LIN {X 0,Y 162.203,Z 311.057,A -85,B 0,C 180,E1 -23302.53,E2 -23302.53} C_VEL
LIN {X 0,Y 161.888,Z 311.469,A -85,B 0,C 180,E1 -23307.51,E2 -23307.51} C_VEL
LIN {X 0,Y 161.935,Z 311.109,A -85,B 0,C 180,E1 -23309.998,E2 -23309.998} C_VEL
LIN {X 0,Y 162.113,Z 310.364,A -85,B 0,C 180,E1 -23312.483,E2 -23312.483} C_VEL
LIN {X 0,Y 162.905,Z 307.824,A -85,B 0,C 180,E1 -23317.126,E2 -23317.126} C_VEL
LIN {X 0,Y 164.1,Z 304.438,A -85,B 0,C 180,E1 -23321.109,E2 -23321.109} C_VEL
LIN {X 0,Y 165.769,Z 300.216,A -85,B 0,C 180,E1 -23324.734,E2 -23324.734} C_VEL
LIN {X 0,Y 168.468,Z 293.815,A -85,B 0,C 180,E1 -23328.86,E2 -23328.86} C_VEL
LIN {X 0,Y 171.418,Z 286.794,A -85,B 0,C 180,E1 -23332.283,E2 -23332.283} C_VEL
LIN {X 0,Y 174.792,Z 278.034,A -85,B 0,C 180,E1 -23335.606,E2 -23335.606} C_VEL
LIN {X 0,Y 178.001,Z 269.053,A -85,B 0,C 180,E1 -23338.277,E2 -23338.277} C_VEL
LIN {X 0,Y 179.645,Z 263.969,A -85,B 0,C 180,E1 -23339.551,E2 -23339.551} C_VEL
LIN {X 0,Y 179.703,Z 256.737,A -85,B 0,C 180,E1 -23341.534,E2 -23341.534} C_VEL
LIN {X 0,Y 178.862,Z 247.409,A -85,B 0,C 180,E1 -23343.952,E2 -23343.952} C_VEL
LIN {X 0,Y 177.345,Z 238.085,A -85,B 0,C 180,E1 -23346.202,E2 -23346.202} C_VEL
LIN {X 0,Y 174.11,Z 227.135,A -85,B 0,C 180,E1 -23348.872,E2 -23348.872} C_VEL
LIN {X 0,Y 169.319,Z 216.684,A -85,B 0,C 180,E1 -23351.656,E2 -23351.656} C_VEL
LIN {X 0,Y 167.341,Z 213.109,A -85,B 0,C 180,E1 -23352.687,E2 -23352.687} C_VEL
LIN {X 0,Y 166.28,Z 211.565,A -85,B 0,C 180,E1 -23353.185,E2 -23353.185} C_VEL
LIN {X 0,Y 164.764,Z 208.871,A -85,B 0,C 180,E1 -23353.961,E2 -23353.961} C_VEL
LIN {X 0,Y 164.403,Z 207.492,A -85,B 0,C 180,E1 -23354.271,E2 -23354.271} C_VEL
LIN {X 0,Y 164.349,Z 207.015,A -85,B 0,C 180,E1 -23356.826,E2 -23356.826} C_VEL
LIN {X 0,Y 164.334,Z 207.015,A -85,B 0,C 180,E1 -23360.328,E2 -23360.328} C_VEL
LIN {X 0,Y 164.319,Z 207.017,A -85,B 0,C 180,E1 -23366.218,E2 -23366.218} C_VEL
LIN {X 0,Y 164.376,Z 207.011,A -85,B 0,C 180,E1 -23369.131,E2 -23369.131} C_VEL
LIN {X 0,Y 164.404,Z 206.998,A -85,B 0,C 180,E1 -23374.691,E2 -23374.691} C_VEL
LIN {X 0,Y 164.507,Z 206.937,A -85,B 0,C 180,E1 -23380.014,E2 -23380.014} C_VEL
LIN {X 0,Y 164.546,Z 206.988,A -85,B 0,C 180,E1 -23385.151,E2 -23385.151} C_VEL
LIN {X 0,Y 164.838,Z 206.938,A -85,B 0,C 180,E1 -23390.18,E2 -23390.18} C_VEL
LIN {X 0,Y 164.846,Z 206.951,A -85,B 0,C 180,E1 -23392.651,E2 -23392.651} C_VEL
LIN {X 0,Y 165.029,Z 206.916,A -85,B 0,C 180,E1 -23397.559,E2 -23397.559} C_VEL
LIN {X 0,Y 165.272,Z 206.899,A -85,B 0,C 180,E1 -23399.999,E2 -23399.999} C_VEL
LIN {X 0,Y 164.763,Z 206.961,A -85,B 0,C 180,E1 -23404.893,E2 -23404.893} C_VEL
LIN {X 0,Y 164.833,Z 206.953,A -85,B 0,C 180,E1 -23407.348,E2 -23407.348} C_VEL
LIN {X 0,Y 164.725,Z 206.968,A -85,B 0,C 180,E1 -23411.13,E2 -23411.13} C_VEL
LIN {X 0,Y 164.485,Z 206.999,A -85,B 0,C 180,E1 -23417.403,E2 -23417.403} C_VEL
LIN {X 0,Y 164.506,Z 206.995,A -85,B 0,C 180,E1 -23419.985,E2 -23419.985} C_VEL
LIN {X 0,Y 164.379,Z 207.01,A -85,B 0,C 180,E1 -23426.135,E2 -23426.135} C_VEL
LIN {X 0,Y 164.37,Z 207.132,A -85,B 0,C 180,E1 -23431.687,E2 -23431.687} C_VEL
LIN {X 0,Y 164.77,Z 209.517,A -85,B 0,C 180,E1 -23436.665,E2 -23436.665} C_VEL
LIN {X 0,Y 165.051,Z 211.251,A -85,B 0,C 180,E1 -23439.971,E2 -23439.971} C_VEL
LIN {X 0,Y 165.48,Z 213.632,A -85,B 0,C 180,E1 -23444.186,E2 -23444.186} C_VEL
LIN {X 0,Y 166.572,Z 216.701,A -85,B 0,C 180,E1 -23444.816,E2 -23444.816} C_VEL
LIN {X 0,Y 168.249,Z 219.242,A -85,B 0,C 180,E1 -23445.593,E2 -23445.593} C_VEL
LIN {X 0,Y 170.168,Z 223.121,A -85,B 0,C 180,E1 -23446.592,E2 -23446.592} C_VEL
LIN {X 0,Y 173.545,Z 231.047,A -85,B 0,C 180,E1 -23448.52,E2 -23448.52} C_VEL
LIN {X 0,Y 175.71,Z 238.733,A -85,B 0,C 180,E1 -23450.216,E2 -23450.216} C_VEL
LIN {X 0,Y 177.253,Z 249.396,A -85,B 0,C 180,E1 -23452.465,E2 -23452.465} C_VEL
LIN {X 0,Y 177.858,Z 259.284,A -85,B 0,C 180,E1 -23454.703,E2 -23454.703} C_VEL
LIN {X 0,Y 177.686,Z 268.748,A -85,B 0,C 180,E1 -23457.058,E2 -23457.058} C_VEL
LIN {X 0,Y 176.797,Z 277.668,A -85,B 0,C 180,E1 -23459.551,E2 -23459.551} C_VEL
LIN {X 0,Y 173.444,Z 286.731,A -85,B 0,C 180,E1 -23462.23,E2 -23462.23} C_VEL
LIN {X 0,Y 170.179,Z 295.589,A -85,B 0,C 180,E1 -23465.612,E2 -23465.612} C_VEL
LIN {X 0,Y 167.31,Z 302.673,A -85,B 0,C 180,E1 -23469.084,E2 -23469.084} C_VEL
LIN {X 0,Y 164.995,Z 308.331,A -85,B 0,C 180,E1 -23472.655,E2 -23472.655} C_VEL
LIN {X 0,Y 163.395,Z 312.791,A -85,B 0,C 180,E1 -23476.319,E2 -23476.319} C_VEL
LIN {X 0,Y 162.403,Z 316.172,A -85,B 0,C 180,E1 -23480.034,E2 -23480.034} C_VEL
LIN {X 0,Y 161.999,Z 317.853,A -85,B 0,C 180,E1 -23482.524,E2 -23482.524} C_VEL
LIN {X 0,Y 161.79,Z 319.131,A -85,B 0,C 180,E1 -23485.018,E2 -23485.018} C_VEL
LIN {X 0,Y 161.765,Z 320.074,A -85,B 0,C 180,E1 -23487.78,E2 -23487.78} C_VEL
LIN {X 0,Y 161.896,Z 320.453,A -85,B 0,C 180,E1 -23490.002,E2 -23490.002} C_VEL
LIN {X 0,Y 161.765,Z 320.488,A -85,B 0,C 180,E1 -23492.492,E2 -23492.492} C_VEL
LIN {X 0,Y 161.791,Z 320.137,A -85,B 0,C 180,E1 -23494.985,E2 -23494.985} C_VEL
LIN {X 0,Y 162.002,Z 319.402,A -85,B 0,C 180,E1 -23497.479,E2 -23497.479} C_VEL
LIN {X 0,Y 162.416,Z 318.234,A -85,B 0,C 180,E1 -23499.968,E2 -23499.968} C_VEL
LIN {X 0,Y 163.497,Z 315.722,A -85,B 0,C 180,E1 -23503.676,E2 -23503.676} C_VEL
LIN {X 0,Y 165.117,Z 312.206,A -85,B 0,C 180,E1 -23507.335,E2 -23507.335} C_VEL
LIN {X 0,Y 167.532,Z 307.605,A -85,B 0,C 180,E1 -23510.89,E2 -23510.89} C_VEL
LIN {X 0,Y 171.01,Z 300.727,A -85,B 0,C 180,E1 -23514.869,E2 -23514.869} C_VEL
LIN {X 0,Y 174.459,Z 293.132,A -85,B 0,C 180,E1 -23518.251,E2 -23518.251} C_VEL
LIN {X 0,Y 178.393,Z 284.443,A -85,B 0,C 180,E1 -23521.198,E2 -23521.198} C_VEL
LIN {X 0,Y 179.136,Z 281.733,A -85,B 0,C 180,E1 -23522.062,E2 -23522.062} C_VEL
LIN {X 0,Y 178.984,Z 277.803,A -85,B 0,C 180,E1 -23523.47,E2 -23523.47} C_VEL
LIN {X 0,Y 177.92,Z 274.075,A -85,B 0,C 180,E1 -23524.927,E2 -23524.927} C_VEL
LIN {X 0,Y 175.412,Z 266.243,A -85,B 0,C 180,E1 -23527.891,E2 -23527.891} C_VEL
LIN {X 0,Y 175.084,Z 263.3,A -85,B 0,C 180,E1 -23528.808,E2 -23528.808} C_VEL
LIN {X 0,Y 174.738,Z 253.125,A -85,B 0,C 180,E1 -23531.496,E2 -23531.496} C_VEL
LIN {X 0,Y 173.737,Z 246.452,A -85,B 0,C 180,E1 -23533.27,E2 -23533.27} C_VEL
LIN {X 0,Y 171.827,Z 240.22,A -85,B 0,C 180,E1 -23535.125,E2 -23535.125} C_VEL
LIN {X 0,Y 168.637,Z 232.567,A -85,B 0,C 180,E1 -23537.626,E2 -23537.626} C_VEL
LIN {X 0,Y 166.729,Z 228.56,A -85,B 0,C 180,E1 -23539.007,E2 -23539.007} C_VEL
LIN {X 0,Y 164.338,Z 223.902,A -85,B 0,C 180,E1 -23540.694,E2 -23540.694} C_VEL
LIN {X 0,Y 162.287,Z 220.406,A -85,B 0,C 180,E1 -23542.092,E2 -23542.092} C_VEL
LIN {X 0,Y 161.446,Z 218.634,A -85,B 0,C 180,E1 -23542.707,E2 -23542.707} C_VEL
LIN {X 0,Y 159.069,Z 215.483,A -85,B 0,C 180,E1 -23544.252,E2 -23544.252} C_VEL
LIN {X 0,Y 158.095,Z 212.845,A -85,B 0,C 180,E1 -23545.087,E2 -23545.087} C_VEL
LIN {X 0,Y 157.947,Z 211.689,A -85,B 0,C 180,E1 -23547.728,E2 -23547.728} C_VEL
LIN {X 0,Y 157.59,Z 209.431,A -85,B 0,C 180,E1 -23553.515,E2 -23553.515} C_VEL
LIN {X 0,Y 157.415,Z 208.47,A -85,B 0,C 180,E1 -23556.309,E2 -23556.309} C_VEL
LIN {X 0,Y 157.441,Z 207.873,A -85,B 0,C 180,E1 -23559.616,E2 -23559.616} C_VEL
LIN {X 0,Y 157.456,Z 207.873,A -85,B 0,C 180,E1 -23564.467,E2 -23564.467} C_VEL
LIN {X 0,Y 157.681,Z 207.842,A -85,B 0,C 180,E1 -23569.731,E2 -23569.731} C_VEL
LIN {X 0,Y 157.758,Z 207.832,A -85,B 0,C 180,E1 -23572.32,E2 -23572.32} C_VEL
LIN {X 0,Y 158.242,Z 207.772,A -85,B 0,C 180,E1 -23580.001,E2 -23580.001} C_VEL
LIN {X 0,Y 157.711,Z 207.84,A -85,B 0,C 180,E1 -23585.114,E2 -23585.114} C_VEL
LIN {X 0,Y 157.756,Z 207.835,A -85,B 0,C 180,E1 -23587.681,E2 -23587.681} C_VEL
LIN {X 0,Y 157.626,Z 207.85,A -85,B 0,C 180,E1 -23591.227,E2 -23591.227} C_VEL
LIN {X 0,Y 157.431,Z 207.873,A -85,B 0,C 180,E1 -23595.537,E2 -23595.537} C_VEL
LIN {X 0,Y 157.364,Z 207.884,A -85,B 0,C 180,E1 -23600.934,E2 -23600.934} C_VEL
LIN {X 0,Y 157.306,Z 207.889,A -85,B 0,C 180,E1 -23606.682,E2 -23606.682} C_VEL
LIN {X 0,Y 157.312,Z 208.05,A -85,B 0,C 180,E1 -23611.918,E2 -23611.918} C_VEL
LIN {X 0,Y 157.324,Z 208.308,A -85,B 0,C 180,E1 -23612.607,E2 -23612.607} C_VEL
LIN {X 0,Y 158.283,Z 210.846,A -85,B 0,C 180,E1 -23613.427,E2 -23613.427} C_VEL
LIN {X 0,Y 160.753,Z 213.678,A -85,B 0,C 180,E1 -23615.039,E2 -23615.039} C_VEL
LIN {X 0,Y 163.069,Z 217.809,A -85,B 0,C 180,E1 -23616.717,E2 -23616.717} C_VEL
LIN {X 0,Y 164.239,Z 219.482,A -85,B 0,C 180,E1 -23617.478,E2 -23617.478} C_VEL
LIN {X 0,Y 166.404,Z 223.337,A -85,B 0,C 180,E1 -23619.019,E2 -23619.019} C_VEL
LIN {X 0,Y 171.596,Z 234.254,A -85,B 0,C 180,E1 -23622.965,E2 -23622.965} C_VEL
LIN {X 0,Y 173.907,Z 240.964,A -85,B 0,C 180,E1 -23625.142,E2 -23625.142} C_VEL
LIN {X 0,Y 175.503,Z 248.167,A -85,B 0,C 180,E1 -23627.335,E2 -23627.335} C_VEL
LIN {X 0,Y 176.566,Z 257.323,A -85,B 0,C 180,E1 -23630.091,E2 -23630.091} C_VEL
LIN {X 0,Y 176.728,Z 265.588,A -85,B 0,C 180,E1 -23632.689,E2 -23632.689} C_VEL
LIN {X 0,Y 176.42,Z 269.664,A -85,B 0,C 180,E1 -23634.015,E2 -23634.015} C_VEL
LIN {X 0,Y 172.646,Z 278.623,A -85,B 0,C 180,E1 -23636.664,E2 -23636.664} C_VEL
LIN {X 0,Y 168.441,Z 287.36,A -85,B 0,C 180,E1 -23639.955,E2 -23639.955} C_VEL
LIN {X 0,Y 164.622,Z 294.525,A -85,B 0,C 180,E1 -23643.505,E2 -23643.505} C_VEL
LIN {X 0,Y 161.73,Z 299.883,A -85,B 0,C 180,E1 -23646.977,E2 -23646.977} C_VEL
LIN {X 0,Y 159.205,Z 304.249,A -85,B 0,C 180,E1 -23650.665,E2 -23650.665} C_VEL
LIN {X 0,Y 157.287,Z 307.544,A -85,B 0,C 180,E1 -23654.448,E2 -23654.448} C_VEL
LIN {X 0,Y 155.652,Z 310.41,A -85,B 0,C 180,E1 -23659.594,E2 -23659.594} C_VEL
LIN {X 0,Y 155.167,Z 311.244,A -85,B 0,C 180,E1 -23662.189,E2 -23662.189} C_VEL
LIN {X 0,Y 154.798,Z 311.67,A -85,B 0,C 180,E1 -23667.396,E2 -23667.396} C_VEL
LIN {X 0,Y 154.835,Z 311.316,A -85,B 0,C 180,E1 -23669.998,E2 -23669.998} C_VEL
LIN {X 0,Y 155.035,Z 310.579,A -85,B 0,C 180,E1 -23672.596,E2 -23672.596} C_VEL
LIN {X 0,Y 155.736,Z 308.452,A -85,B 0,C 180,E1 -23676.869,E2 -23676.869} C_VEL
LIN {X 0,Y 157.159,Z 304.68,A -85,B 0,C 180,E1 -23681.607,E2 -23681.607} C_VEL
LIN {X 0,Y 158.921,Z 300.471,A -85,B 0,C 180,E1 -23685.384,E2 -23685.384} C_VEL
LIN {X 0,Y 161.764,Z 294.086,A -85,B 0,C 180,E1 -23689.673,E2 -23689.673} C_VEL
LIN {X 0,Y 164.871,Z 287.089,A -85,B 0,C 180,E1 -23693.219,E2 -23693.219} C_VEL
LIN {X 0,Y 168.434,Z 278.348,A -85,B 0,C 180,E1 -23696.647,E2 -23696.647} C_VEL
LIN {X 0,Y 171.792,Z 269.391,A -85,B 0,C 180,E1 -23699.397,E2 -23699.397} C_VEL
LIN {X 0,Y 173.31,Z 264.918,A -85,B 0,C 180,E1 -23700.556,E2 -23700.556} C_VEL
LIN {X 0,Y 173.334,Z 256.195,A -85,B 0,C 180,E1 -23703.096,E2 -23703.096} C_VEL
LIN {X 0,Y 172.301,Z 245.415,A -85,B 0,C 180,E1 -23706.01,E2 -23706.01} C_VEL
LIN {X 0,Y 170.636,Z 237.194,A -85,B 0,C 180,E1 -23708.151,E2 -23708.151} C_VEL
LIN {X 0,Y 168.166,Z 229.23,A -85,B 0,C 180,E1 -23710.296,E2 -23710.296} C_VEL
LIN {X 0,Y 163.955,Z 220.22,A -85,B 0,C 180,E1 -23712.995,E2 -23712.995} C_VEL
LIN {X 0,Y 162.101,Z 216.724,A -85,B 0,C 180,E1 -23714.084,E2 -23714.084} C_VEL
LIN {X 0,Y 160.266,Z 213.131,A -85,B 0,C 180,E1 -23715.181,E2 -23715.181} C_VEL
LIN {X 0,Y 157.998,Z 210.26,A -85,B 0,C 180,E1 -23716.352,E2 -23716.352} C_VEL
LIN {X 0,Y 157.297,Z 207.894,A -85,B 0,C 180,E1 -23716.889,E2 -23716.889} C_VEL
LIN {X 0,Y 157.252,Z 207.899,A -85,B 0,C 180,E1 -23721.266,E2 -23721.266} C_VEL
LIN {X 0,Y 157.278,Z 207.892,A -85,B 0,C 180,E1 -23724.485,E2 -23724.485} C_VEL
LIN {X 0,Y 157.282,Z 207.89,A -85,B 0,C 180,E1 -23728.093,E2 -23728.093} C_VEL
LIN {X 0,Y 157.308,Z 207.89,A -85,B 0,C 180,E1 -23733.463,E2 -23733.463} C_VEL
LIN {X 0,Y 157.433,Z 207.815,A -85,B 0,C 180,E1 -23739.614,E2 -23739.614} C_VEL
LIN {X 0,Y 157.474,Z 207.865,A -85,B 0,C 180,E1 -23744.467,E2 -23744.467} C_VEL
LIN {X 0,Y 157.757,Z 207.818,A -85,B 0,C 180,E1 -23749.735,E2 -23749.735} C_VEL
LIN {X 0,Y 157.808,Z 207.828,A -85,B 0,C 180,E1 -23752.321,E2 -23752.321} C_VEL
LIN {X 0,Y 158.235,Z 207.775,A -85,B 0,C 180,E1 -23759.999,E2 -23759.999} C_VEL
LIN {X 0,Y 157.712,Z 207.84,A -85,B 0,C 180,E1 -23765.113,E2 -23765.113} C_VEL
LIN {X 0,Y 157.79,Z 207.832,A -85,B 0,C 180,E1 -23767.678,E2 -23767.678} C_VEL
LIN {X 0,Y 157.656,Z 207.848,A -85,B 0,C 180,E1 -23771.299,E2 -23771.299} C_VEL
LIN {X 0,Y 157.443,Z 207.876,A -85,B 0,C 180,E1 -23775.535,E2 -23775.535} C_VEL
LIN {X 0,Y 157.401,Z 207.879,A -85,B 0,C 180,E1 -23780.928,E2 -23780.928} C_VEL
LIN {X 0,Y 157.301,Z 207.89,A -85,B 0,C 180,E1 -23786.686,E2 -23786.686} C_VEL
LIN {X 0,Y 157.31,Z 207.905,A -85,B 0,C 180,E1 -23790.08,E2 -23790.08} C_VEL
LIN {X 0,Y 157.7,Z 210.271,A -85,B 0,C 180,E1 -23795.405,E2 -23795.405} C_VEL
LIN {X 0,Y 158.195,Z 213.385,A -85,B 0,C 180,E1 -23801.502,E2 -23801.502} C_VEL
LIN {X 0,Y 159.386,Z 216.528,A -85,B 0,C 180,E1 -23802.255,E2 -23802.255} C_VEL
LIN {X 0,Y 161.229,Z 219.165,A -85,B 0,C 180,E1 -23803.199,E2 -23803.199} C_VEL
LIN {X 0,Y 163.297,Z 223.265,A -85,B 0,C 180,E1 -23804.393,E2 -23804.393} C_VEL
LIN {X 0,Y 166.774,Z 230.949,A -85,B 0,C 180,E1 -23806.52,E2 -23806.52} C_VEL
LIN {X 0,Y 169.541,Z 239.112,A -85,B 0,C 180,E1 -23808.62,E2 -23808.62} C_VEL
LIN {X 0,Y 170.958,Z 248.36,A -85,B 0,C 180,E1 -23810.71,E2 -23810.71} C_VEL
LIN {X 0,Y 171.59,Z 258.978,A -85,B 0,C 180,E1 -23813.236,E2 -23813.236} C_VEL
LIN {X 0,Y 171.422,Z 268.343,A -85,B 0,C 180,E1 -23815.681,E2 -23815.681} C_VEL
LIN {X 0,Y 170.445,Z 277.327,A -85,B 0,C 180,E1 -23818.287,E2 -23818.287} C_VEL
LIN {X 0,Y 168.499,Z 283,A -85,B 0,C 180,E1 -23819.97,E2 -23819.97} C_VEL
LIN {X 0,Y 165.319,Z 291.103,A -85,B 0,C 180,E1 -23822.811,E2 -23822.811} C_VEL
LIN {X 0,Y 162.159,Z 299.059,A -85,B 0,C 180,E1 -23826.369,E2 -23826.369} C_VEL
LIN {X 0,Y 159.836,Z 304.439,A -85,B 0,C 180,E1 -23829.408,E2 -23829.408} C_VEL
LIN {X 0,Y 157.544,Z 309.705,A -85,B 0,C 180,E1 -23833.147,E2 -23833.147} C_VEL
LIN {X 0,Y 156.046,Z 313.804,A -85,B 0,C 180,E1 -23836.989,E2 -23836.989} C_VEL
LIN {X 0,Y 155.406,Z 315.944,A -85,B 0,C 180,E1 -23839.581,E2 -23839.581} C_VEL
LIN {X 0,Y 154.948,Z 317.631,A -85,B 0,C 180,E1 -23842.182,E2 -23842.182} C_VEL
LIN {X 0,Y 154.71,Z 318.914,A -85,B 0,C 180,E1 -23844.789,E2 -23844.789} C_VEL
LIN {X 0,Y 154.683,Z 319.986,A -85,B 0,C 180,E1 -23848.307,E2 -23848.307} C_VEL
LIN {X 0,Y 154.794,Z 320.253,A -85,B 0,C 180,E1 -23850.002,E2 -23850.002} C_VEL
LIN {X 0,Y 154.69,Z 320.293,A -85,B 0,C 180,E1 -23852.606,E2 -23852.606} C_VEL
LIN {X 0,Y 154.952,Z 319.218,A -85,B 0,C 180,E1 -23857.822,E2 -23857.822} C_VEL
LIN {X 0,Y 155.418,Z 318.06,A -85,B 0,C 180,E1 -23860.422,E2 -23860.422} C_VEL
LIN {X 0,Y 156.133,Z 316.478,A -85,B 0,C 180,E1 -23863.007,E2 -23863.007} C_VEL
LIN {X 0,Y 157.659,Z 313.312,A -85,B 0,C 180,E1 -23866.844,E2 -23866.844} C_VEL
LIN {X 0,Y 159.989,Z 309.096,A -85,B 0,C 180,E1 -23870.575,E2 -23870.575} C_VEL
LIN {X 0,Y 162.92,Z 303.71,A -85,B 0,C 180,E1 -23874.193,E2 -23874.193} C_VEL
LIN {X 0,Y 166.299,Z 296.973,A -85,B 0,C 180,E1 -23877.702,E2 -23877.702} C_VEL
LIN {X 0,Y 170.363,Z 288.626,A -85,B 0,C 180,E1 -23881.041,E2 -23881.041} C_VEL
LIN {X 0,Y 173.344,Z 281.875,A -85,B 0,C 180,E1 -23883.184,E2 -23883.184} C_VEL
LIN {X 0,Y 174.641,Z 273.581,A -85,B 0,C 180,E1 -23885.819,E2 -23885.819} C_VEL
LIN {X 0,Y 175.094,Z 264.082,A -85,B 0,C 180,E1 -23888.583,E2 -23888.583} C_VEL
LIN {X 0,Y 175.084,Z 263.3,A -85,B 0,C 180,E1 -23888.808,E2 -23888.808} C_VEL
LIN {X 0,Y 174.426,Z 259.081,A -85,B 0,C 180,E1 -23890.152,E2 -23890.152} C_VEL
LIN {X 0,Y 172.876,Z 255.276,A -85,B 0,C 180,E1 -23891.575,E2 -23891.575} C_VEL
LIN {X 0,Y 168.701,Z 248.158,A -85,B 0,C 180,E1 -23894.542,E2 -23894.542} C_VEL
LIN {X 0,Y 166.316,Z 242.998,A -85,B 0,C 180,E1 -23896.51,E2 -23896.51} C_VEL
LIN {X 0,Y 162.824,Z 234.197,A -85,B 0,C 180,E1 -23899.651,E2 -23899.651} C_VEL
LIN {X 0,Y 159.954,Z 228.545,A -85,B 0,C 180,E1 -23901.939,E2 -23901.939} C_VEL
LIN {X 0,Y 157.693,Z 224.076,A -85,B 0,C 180,E1 -23903.785,E2 -23903.785} C_VEL
LIN {X 0,Y 155.296,Z 220.209,A -85,B 0,C 180,E1 -23905.648,E2 -23905.648} C_VEL
LIN {X 0,Y 154.514,Z 218.494,A -85,B 0,C 180,E1 -23906.335,E2 -23906.335} C_VEL
LIN {X 0,Y 152.056,Z 215.517,A -85,B 0,C 180,E1 -23908.204,E2 -23908.204} C_VEL
LIN {X 0,Y 150.93,Z 212.808,A -85,B 0,C 180,E1 -23909.286,E2 -23909.286} C_VEL
LIN {X 0,Y 150.85,Z 212.305,A -85,B 0,C 180,E1 -23909.945,E2 -23909.945} C_VEL
LIN {X 0,Y 150.531,Z 210.458,A -85,B 0,C 180,E1 -23915.154,E2 -23915.154} C_VEL
LIN {X 0,Y 150.387,Z 208.751,A -85,B 0,C 180,E1 -23920.906,E2 -23920.906} C_VEL
LIN {X 0,Y 150.432,Z 208.748,A -85,B 0,C 180,E1 -23926.492,E2 -23926.492} C_VEL
LIN {X 0,Y 150.604,Z 208.726,A -85,B 0,C 180,E1 -23929.243,E2 -23929.243} C_VEL
LIN {X 0,Y 150.695,Z 208.713,A -85,B 0,C 180,E1 -23931.958,E2 -23931.958} C_VEL
LIN {X 0,Y 151.204,Z 208.649,A -85,B 0,C 180,E1 -23940.001,E2 -23940.001} C_VEL
LIN {X 0,Y 150.64,Z 208.716,A -85,B 0,C 180,E1 -23946.982,E2 -23946.982} C_VEL
LIN {X 0,Y 150.568,Z 208.728,A -85,B 0,C 180,E1 -23951.43,E2 -23951.43} C_VEL
LIN {X 0,Y 150.343,Z 208.758,A -85,B 0,C 180,E1 -23956.289,E2 -23956.289} C_VEL
LIN {X 0,Y 150.346,Z 208.758,A -85,B 0,C 180,E1 -23960.792,E2 -23960.792} C_VEL
LIN {X 0,Y 150.238,Z 208.771,A -85,B 0,C 180,E1 -23967.281,E2 -23967.281} C_VEL
LIN {X 0,Y 150.203,Z 208.777,A -85,B 0,C 180,E1 -23968.279,E2 -23968.279} C_VEL
LIN {X 0,Y 150.914,Z 211.097,A -85,B 0,C 180,E1 -23969.084,E2 -23969.084} C_VEL
LIN {X 0,Y 152.923,Z 213.602,A -85,B 0,C 180,E1 -23970.723,E2 -23970.723} C_VEL
LIN {X 0,Y 154.214,Z 214.632,A -85,B 0,C 180,E1 -23971.641,E2 -23971.641} C_VEL
LIN {X 0,Y 156.009,Z 218.019,A -85,B 0,C 180,E1 -23973.205,E2 -23973.205} C_VEL
LIN {X 0,Y 157.587,Z 220.032,A -85,B 0,C 180,E1 -23974.364,E2 -23974.364} C_VEL
LIN {X 0,Y 159.667,Z 223.754,A -85,B 0,C 180,E1 -23976.067,E2 -23976.067} C_VEL
LIN {X 0,Y 163.659,Z 231.631,A -85,B 0,C 180,E1 -23979.381,E2 -23979.381} C_VEL
LIN {X 0,Y 166.926,Z 239.317,A -85,B 0,C 180,E1 -23982.35,E2 -23982.35} C_VEL
LIN {X 0,Y 169.117,Z 247.172,A -85,B 0,C 180,E1 -23985.054,E2 -23985.054} C_VEL
LIN {X 0,Y 170.207,Z 254.802,A -85,B 0,C 180,E1 -23987.505,E2 -23987.505} C_VEL
LIN {X 0,Y 170.646,Z 263.364,A -85,B 0,C 180,E1 -23990.333,E2 -23990.333} C_VEL
LIN {X 0,Y 170.321,Z 270.371,A -85,B 0,C 180,E1 -23992.758,E2 -23992.758} C_VEL
LIN {X 0,Y 167.564,Z 277.078,A -85,B 0,C 180,E1 -23994.782,E2 -23994.782} C_VEL
LIN {X 0,Y 163.02,Z 286.111,A -85,B 0,C 180,E1 -23998.123,E2 -23998.123} C_VEL
LIN {X 0,Y 158.942,Z 293.494,A -85,B 0,C 180,E1 -24001.691,E2 -24001.691} C_VEL
LIN {X 0,Y 155.173,Z 300.024,A -85,B 0,C 180,E1 -24005.944,E2 -24005.944} C_VEL
LIN {X 0,Y 152.509,Z 304.402,A -85,B 0,C 180,E1 -24009.78,E2 -24009.78} C_VEL
LIN {X 0,Y 150.432,Z 307.711,A -85,B 0,C 180,E1 -24013.72,E2 -24013.72} C_VEL
LIN {X 0,Y 148.664,Z 310.588,A -85,B 0,C 180,E1 -24019.099,E2 -24019.099} C_VEL
LIN {X 0,Y 148.113,Z 311.431,A -85,B 0,C 180,E1 -24021.815,E2 -24021.815} C_VEL
LIN {X 0,Y 147.718,Z 311.87,A -85,B 0,C 180,E1 -24027.271,E2 -24027.271} C_VEL
LIN {X 0,Y 147.748,Z 311.522,A -85,B 0,C 180,E1 -24029.998,E2 -24029.998} C_VEL
LIN {X 0,Y 147.946,Z 310.793,A -85,B 0,C 180,E1 -24032.721,E2 -24032.721} C_VEL
LIN {X 0,Y 148.54,Z 309.074,A -85,B 0,C 180,E1 -24036.482,E2 -24036.482} C_VEL
LIN {X 0,Y 150.216,Z 304.922,A -85,B 0,C 180,E1 -24042.151,E2 -24042.151} C_VEL
LIN {X 0,Y 152.105,Z 300.727,A -85,B 0,C 180,E1 -24046.092,E2 -24046.092} C_VEL
LIN {X 0,Y 155.096,Z 294.356,A -85,B 0,C 180,E1 -24050.556,E2 -24050.556} C_VEL
LIN {X 0,Y 158.382,Z 287.384,A -85,B 0,C 180,E1 -24054.23,E2 -24054.23} C_VEL
LIN {X 0,Y 162.115,Z 278.664,A -85,B 0,C 180,E1 -24057.773,E2 -24057.773} C_VEL
LIN {X 0,Y 165.656,Z 269.729,A -85,B 0,C 180,E1 -24060.6,E2 -24060.6} C_VEL
LIN {X 0,Y 166.986,Z 265.869,A -85,B 0,C 180,E1 -24061.647,E2 -24061.647} C_VEL
LIN {X 0,Y 167.052,Z 255.964,A -85,B 0,C 180,E1 -24064.697,E2 -24064.697} C_VEL
LIN {X 0,Y 166.044,Z 245.62,A -85,B 0,C 180,E1 -24067.66,E2 -24067.66} C_VEL
LIN {X 0,Y 163.914,Z 236.216,A -85,B 0,C 180,E1 -24070.346,E2 -24070.346} C_VEL
LIN {X 0,Y 160.826,Z 228.089,A -85,B 0,C 180,E1 -24072.875,E2 -24072.875} C_VEL
LIN {X 0,Y 157.75,Z 221.69,A -85,B 0,C 180,E1 -24075.027,E2 -24075.027} C_VEL
LIN {X 0,Y 155.572,Z 217.717,A -85,B 0,C 180,E1 -24076.454,E2 -24076.454} C_VEL
LIN {X 0,Y 153.648,Z 214.551,A -85,B 0,C 180,E1 -24077.682,E2 -24077.682} C_VEL
LIN {X 0,Y 153.02,Z 213.601,A -85,B 0,C 180,E1 -24078.069,E2 -24078.069} C_VEL
LIN {X 0,Y 150.999,Z 211.254,A -85,B 0,C 180,E1 -24079.24,E2 -24079.24} C_VEL
LIN {X 0,Y 150.194,Z 208.776,A -85,B 0,C 180,E1 -24079.953,E2 -24079.953} C_VEL
LIN {X 0,Y 150.21,Z 208.773,A -85,B 0,C 180,E1 -24082.684,E2 -24082.684} C_VEL
LIN {X 0,Y 150.205,Z 208.771,A -85,B 0,C 180,E1 -24087.364,E2 -24087.364} C_VEL
LIN {X 0,Y 150.232,Z 208.772,A -85,B 0,C 180,E1 -24092.716,E2 -24092.716} C_VEL
LIN {X 0,Y 150.377,Z 208.691,A -85,B 0,C 180,E1 -24099.167,E2 -24099.167} C_VEL
LIN {X 0,Y 150.383,Z 208.74,A -85,B 0,C 180,E1 -24103.715,E2 -24103.715} C_VEL
LIN {X 0,Y 150.674,Z 208.699,A -85,B 0,C 180,E1 -24109.246,E2 -24109.246} C_VEL
LIN {X 0,Y 150.747,Z 208.705,A -85,B 0,C 180,E1 -24111.959,E2 -24111.959} C_VEL
LIN {X 0,Y 151.196,Z 208.652,A -85,B 0,C 180,E1 -24119.999,E2 -24119.999} C_VEL
LIN {X 0,Y 150.661,Z 208.719,A -85,B 0,C 180,E1 -24125.353,E2 -24125.353} C_VEL
LIN {X 0,Y 150.725,Z 208.712,A -85,B 0,C 180,E1 -24128.041,E2 -24128.041} C_VEL
LIN {X 0,Y 150.59,Z 208.728,A -85,B 0,C 180,E1 -24131.488,E2 -24131.488} C_VEL
LIN {X 0,Y 150.356,Z 208.757,A -85,B 0,C 180,E1 -24136.287,E2 -24136.287} C_VEL
LIN {X 0,Y 150.376,Z 208.754,A -85,B 0,C 180,E1 -24140.832,E2 -24140.832} C_VEL
LIN {X 0,Y 150.231,Z 208.772,A -85,B 0,C 180,E1 -24147.283,E2 -24147.283} C_VEL
LIN {X 0,Y 150.206,Z 208.847,A -85,B 0,C 180,E1 -24148.658,E2 -24148.658} C_VEL
LIN {X 0,Y 150.547,Z 210.529,A -85,B 0,C 180,E1 -24152.839,E2 -24152.839} C_VEL
LIN {X 0,Y 150.92,Z 213.026,A -85,B 0,C 180,E1 -24158.364,E2 -24158.364} C_VEL
LIN {X 0,Y 152.106,Z 216.252,A -85,B 0,C 180,E1 -24159.253,E2 -24159.253} C_VEL
LIN {X 0,Y 154.222,Z 219.149,A -85,B 0,C 180,E1 -24160.477,E2 -24160.477} C_VEL
LIN {X 0,Y 156.099,Z 222.817,A -85,B 0,C 180,E1 -24161.699,E2 -24161.699} C_VEL
LIN {X 0,Y 157.354,Z 225.261,A -85,B 0,C 180,E1 -24162.496,E2 -24162.496} C_VEL
LIN {X 0,Y 160.945,Z 232.932,A -85,B 0,C 180,E1 -24164.941,E2 -24164.941} C_VEL
LIN {X 0,Y 163.837,Z 241.739,A -85,B 0,C 180,E1 -24167.412,E2 -24167.412} C_VEL
LIN {X 0,Y 165.07,Z 250.965,A -85,B 0,C 180,E1 -24169.7,E2 -24169.7} C_VEL
LIN {X 0,Y 165.418,Z 261.952,A -85,B 0,C 180,E1 -24172.518,E2 -24172.518} C_VEL
LIN {X 0,Y 164.895,Z 271.574,A -85,B 0,C 180,E1 -24175.246,E2 -24175.246} C_VEL
LIN {X 0,Y 163.785,Z 278.967,A -85,B 0,C 180,E1 -24177.567,E2 -24177.567} C_VEL
LIN {X 0,Y 160.288,Z 287.755,A -85,B 0,C 180,E1 -24180.449,E2 -24180.449} C_VEL
LIN {X 0,Y 156.893,Z 295.84,A -85,B 0,C 180,E1 -24183.84,E2 -24183.84} C_VEL
LIN {X 0,Y 154.025,Z 302.14,A -85,B 0,C 180,E1 -24187.183,E2 -24187.183} C_VEL
LIN {X 0,Y 151.473,Z 307.829,A -85,B 0,C 180,E1 -24191.051,E2 -24191.051} C_VEL
LIN {X 0,Y 149.57,Z 312.312,A -85,B 0,C 180,E1 -24195.026,E2 -24195.026} C_VEL
LIN {X 0,Y 148.39,Z 315.716,A -85,B 0,C 180,E1 -24199.082,E2 -24199.082} C_VEL
LIN {X 0,Y 147.898,Z 317.409,A -85,B 0,C 180,E1 -24201.807,E2 -24201.807} C_VEL
LIN {X 0,Y 147.633,Z 318.698,A -85,B 0,C 180,E1 -24204.539,E2 -24204.539} C_VEL
LIN {X 0,Y 147.612,Z 319.908,A -85,B 0,C 180,E1 -24208.946,E2 -24208.946} C_VEL
LIN {X 0,Y 147.606,Z 320.098,A -85,B 0,C 180,E1 -24212.731,E2 -24212.731} C_VEL
LIN {X 0,Y 147.902,Z 319.033,A -85,B 0,C 180,E1 -24218.197,E2 -24218.197} C_VEL
LIN {X 0,Y 148.406,Z 317.885,A -85,B 0,C 180,E1 -24220.92,E2 -24220.92} C_VEL
LIN {X 0,Y 149.179,Z 316.309,A -85,B 0,C 180,E1 -24223.625,E2 -24223.625} C_VEL
LIN {X 0,Y 150.86,Z 313.155,A -85,B 0,C 180,E1 -24227.627,E2 -24227.627} C_VEL
LIN {X 0,Y 153.348,Z 308.951,A -85,B 0,C 180,E1 -24231.509,E2 -24231.509} C_VEL
LIN {X 0,Y 156.472,Z 303.578,A -85,B 0,C 180,E1 -24235.258,E2 -24235.258} C_VEL
LIN {X 0,Y 160.028,Z 296.855,A -85,B 0,C 180,E1 -24238.887,E2 -24238.887} C_VEL
LIN {X 0,Y 164.301,Z 288.529,A -85,B 0,C 180,E1 -24242.322,E2 -24242.322} C_VEL
LIN {X 0,Y 166.689,Z 283.578,A -85,B 0,C 180,E1 -24243.962,E2 -24243.962} C_VEL
LIN {X 0,Y 167.946,Z 278.002,A -85,B 0,C 180,E1 -24245.862,E2 -24245.862} C_VEL
LIN {X 0,Y 168.887,Z 269.391,A -85,B 0,C 180,E1 -24248.623,E2 -24248.623} C_VEL
LIN {X 0,Y 169.119,Z 258.96,A -85,B 0,C 180,E1 -24251.674,E2 -24251.674} C_VEL
LIN {X 0,Y 168.49,Z 251.064,A -85,B 0,C 180,E1 -24253.912,E2 -24253.912} C_VEL
LIN {X 0,Y 166.844,Z 244.583,A -85,B 0,C 180,E1 -24255.969,E2 -24255.969} C_VEL
LIN {X 0,Y 166.316,Z 242.998,A -85,B 0,C 180,E1 -24256.51,E2 -24256.51} C_VEL
LIN {X 0,Y 164.51,Z 239.362,A -85,B 0,C 180,E1 -24257.99,E2 -24257.99} C_VEL
LIN {X 0,Y 162.082,Z 236.448,A -85,B 0,C 180,E1 -24259.589,E2 -24259.589} C_VEL
LIN {X 0,Y 153.126,Z 228.349,A -85,B 0,C 180,E1 -24265.436,E2 -24265.436} C_VEL
LIN {X 0,Y 151.043,Z 224.175,A -85,B 0,C 180,E1 -24267.453,E2 -24267.453} C_VEL
LIN {X 0,Y 148.619,Z 220.597,A -85,B 0,C 180,E1 -24269.643,E2 -24269.643} C_VEL
LIN {X 0,Y 147.747,Z 218.495,A -85,B 0,C 180,E1 -24270.624,E2 -24270.624} C_VEL
LIN {X 0,Y 144.904,Z 215.32,A -85,B 0,C 180,E1 -24273.293,E2 -24273.293} C_VEL
LIN {X 0,Y 143.777,Z 212.757,A -85,B 0,C 180,E1 -24274.678,E2 -24274.678} C_VEL
LIN {X 0,Y 143.612,Z 212.07,A -85,B 0,C 180,E1 -24275.034,E2 -24275.034} C_VEL
LIN {X 0,Y 143.507,Z 210.599,A -85,B 0,C 180,E1 -24279.952,E2 -24279.952} C_VEL
LIN {X 0,Y 143.347,Z 209.886,A -85,B 0,C 180,E1 -24282.893,E2 -24282.893} C_VEL
LIN {X 0,Y 143.53,Z 209.607,A -85,B 0,C 180,E1 -24288.706,E2 -24288.706} C_VEL
LIN {X 0,Y 143.617,Z 209.596,A -85,B 0,C 180,E1 -24291.559,E2 -24291.559} C_VEL
LIN {X 0,Y 144.163,Z 209.526,A -85,B 0,C 180,E1 -24300.001,E2 -24300.001} C_VEL
LIN {X 0,Y 143.564,Z 209.595,A -85,B 0,C 180,E1 -24306.985,E2 -24306.985} C_VEL
LIN {X 0,Y 143.495,Z 209.608,A -85,B 0,C 180,E1 -24311.619,E2 -24311.619} C_VEL
LIN {X 0,Y 143.287,Z 209.634,A -85,B 0,C 180,E1 -24317.116,E2 -24317.116} C_VEL
LIN {X 0,Y 143.235,Z 209.641,A -85,B 0,C 180,E1 -24322.019,E2 -24322.019} C_VEL
LIN {X 0,Y 143.203,Z 209.867,A -85,B 0,C 180,E1 -24322.912,E2 -24322.912} C_VEL
LIN {X 0,Y 143.914,Z 212.049,A -85,B 0,C 180,E1 -24323.951,E2 -24323.951} C_VEL
LIN {X 0,Y 145.939,Z 214.431,A -85,B 0,C 180,E1 -24326.035,E2 -24326.035} C_VEL
LIN {X 0,Y 147.4,Z 215.474,A -85,B 0,C 180,E1 -24327.324,E2 -24327.324} C_VEL
LIN {X 0,Y 149.044,Z 218.688,A -85,B 0,C 180,E1 -24329.097,E2 -24329.097} C_VEL
LIN {X 0,Y 151.036,Z 220.822,A -85,B 0,C 180,E1 -24330.788,E2 -24330.788} C_VEL
LIN {X 0,Y 153.361,Z 224.795,A -85,B 0,C 180,E1 -24332.97,E2 -24332.97} C_VEL
LIN {X 0,Y 156.812,Z 231.437,A -85,B 0,C 180,E1 -24336.226,E2 -24336.226} C_VEL
LIN {X 0,Y 160.051,Z 238.807,A -85,B 0,C 180,E1 -24339.48,E2 -24339.48} C_VEL
LIN {X 0,Y 162.406,Z 245.313,A -85,B 0,C 180,E1 -24342.128,E2 -24342.128} C_VEL
LIN {X 0,Y 163.974,Z 253.106,A -85,B 0,C 180,E1 -24344.965,E2 -24344.965} C_VEL
LIN {X 0,Y 164.557,Z 262.623,A -85,B 0,C 180,E1 -24348.281,E2 -24348.281} C_VEL
LIN {X 0,Y 164.162,Z 271.302,A -85,B 0,C 180,E1 -24351.457,E2 -24351.457} C_VEL
LIN {X 0,Y 163.336,Z 273.899,A -85,B 0,C 180,E1 -24352.307,E2 -24352.307} C_VEL
LIN {X 0,Y 158.548,Z 283.413,A -85,B 0,C 180,E1 -24355.586,E2 -24355.586} C_VEL
LIN {X 0,Y 154.092,Z 291.272,A -85,B 0,C 180,E1 -24359.13,E2 -24359.13} C_VEL
LIN {X 0,Y 150.789,Z 296.719,A -85,B 0,C 180,E1 -24362.322,E2 -24362.322} C_VEL
LIN {X 0,Y 147.722,Z 301.768,A -85,B 0,C 180,E1 -24366.147,E2 -24366.147} C_VEL
LIN {X 0,Y 144.968,Z 305.792,A -85,B 0,C 180,E1 -24370.162,E2 -24370.162} C_VEL
LIN {X 0,Y 143.582,Z 307.877,A -85,B 0,C 180,E1 -24372.921,E2 -24372.921} C_VEL
LIN {X 0,Y 142.507,Z 309.521,A -85,B 0,C 180,E1 -24375.724,E2 -24375.724} C_VEL
LIN {X 0,Y 141.674,Z 310.766,A -85,B 0,C 180,E1 -24378.554,E2 -24378.554} C_VEL
LIN {X 0,Y 141.072,Z 311.618,A -85,B 0,C 180,E1 -24381.403,E2 -24381.403} C_VEL
LIN {X 0,Y 140.725,Z 312.038,A -85,B 0,C 180,E1 -24384.266,E2 -24384.266} C_VEL
LIN {X 0,Y 140.606,Z 311.969,A -85,B 0,C 180,E1 -24388.568,E2 -24388.568} C_VEL
LIN {X 0,Y 140.866,Z 311.007,A -85,B 0,C 180,E1 -24392.858,E2 -24392.858} C_VEL
LIN {X 0,Y 141.263,Z 309.855,A -85,B 0,C 180,E1 -24395.708,E2 -24395.708} C_VEL
LIN {X 0,Y 141.934,Z 308.293,A -85,B 0,C 180,E1 -24398.54,E2 -24398.54} C_VEL
LIN {X 0,Y 143.305,Z 305.164,A -85,B 0,C 180,E1 -24402.747,E2 -24402.747} C_VEL
LIN {X 0,Y 145.294,Z 300.983,A -85,B 0,C 180,E1 -24406.868,E2 -24406.868} C_VEL
LIN {X 0,Y 148.469,Z 294.626,A -85,B 0,C 180,E1 -24411.518,E2 -24411.518} C_VEL
LIN {X 0,Y 151.956,Z 287.677,A -85,B 0,C 180,E1 -24415.325,E2 -24415.325} C_VEL
LIN {X 0,Y 155.879,Z 278.978,A -85,B 0,C 180,E1 -24418.987,E2 -24418.987} C_VEL
LIN {X 0,Y 159.606,Z 270.066,A -85,B 0,C 180,E1 -24421.893,E2 -24421.893} C_VEL
LIN {X 0,Y 160.511,Z 267.676,A -85,B 0,C 180,E1 -24422.57,E2 -24422.57} C_VEL
LIN {X 0,Y 160.923,Z 261.549,A -85,B 0,C 180,E1 -24424.588,E2 -24424.588} C_VEL
LIN {X 0,Y 160.444,Z 250.852,A -85,B 0,C 180,E1 -24427.957,E2 -24427.957} C_VEL
LIN {X 0,Y 159.254,Z 243.155,A -85,B 0,C 180,E1 -24430.302,E2 -24430.302} C_VEL
LIN {X 0,Y 157.717,Z 237.295,A -85,B 0,C 180,E1 -24432.171,E2 -24432.171} C_VEL
LIN {X 0,Y 154.249,Z 228.574,A -85,B 0,C 180,E1 -24435.233,E2 -24435.233} C_VEL
LIN {X 0,Y 151.345,Z 222.867,A -85,B 0,C 180,E1 -24437.45,E2 -24437.45} C_VEL
LIN {X 0,Y 149.021,Z 219.012,A -85,B 0,C 180,E1 -24439.128,E2 -24439.128} C_VEL
LIN {X 0,Y 147.068,Z 216.151,A -85,B 0,C 180,E1 -24440.492,E2 -24440.492} C_VEL
LIN {X 0,Y 146.263,Z 214.668,A -85,B 0,C 180,E1 -24441.121,E2 -24441.121} C_VEL
LIN {X 0,Y 144.241,Z 212.593,A -85,B 0,C 180,E1 -24442.453,E2 -24442.453} C_VEL
LIN {X 0,Y 143.226,Z 210.153,A -85,B 0,C 180,E1 -24443.335,E2 -24443.335} C_VEL
LIN {X 0,Y 143.126,Z 209.658,A -85,B 0,C 180,E1 -24443.542,E2 -24443.542} C_VEL
LIN {X 0,Y 143.173,Z 209.647,A -85,B 0,C 180,E1 -24447.318,E2 -24447.318} C_VEL
LIN {X 0,Y 143.15,Z 209.651,A -85,B 0,C 180,E1 -24453.777,E2 -24453.777} C_VEL
LIN {X 0,Y 143.331,Z 209.568,A -85,B 0,C 180,E1 -24459.925,E2 -24459.925} C_VEL
LIN {X 0,Y 143.373,Z 209.626,A -85,B 0,C 180,E1 -24465.812,E2 -24465.812} C_VEL
LIN {X 0,Y 143.588,Z 209.581,A -85,B 0,C 180,E1 -24468.709,E2 -24468.709} C_VEL
LIN {X 0,Y 143.669,Z 209.585,A -85,B 0,C 180,E1 -24471.56,E2 -24471.56} C_VEL
LIN {X 0,Y 144.156,Z 209.529,A -85,B 0,C 180,E1 -24479.999,E2 -24479.999} C_VEL
LIN {X 0,Y 143.608,Z 209.598,A -85,B 0,C 180,E1 -24485.616,E2 -24485.616} C_VEL
LIN {X 0,Y 143.644,Z 209.593,A -85,B 0,C 180,E1 -24488.44,E2 -24488.44} C_VEL
LIN {X 0,Y 143.534,Z 209.606,A -85,B 0,C 180,E1 -24491.713,E2 -24491.713} C_VEL
LIN {X 0,Y 143.302,Z 209.636,A -85,B 0,C 180,E1 -24497.113,E2 -24497.113} C_VEL
LIN {X 0,Y 143.297,Z 209.636,A -85,B 0,C 180,E1 -24501.29,E2 -24501.29} C_VEL
LIN {X 0,Y 143.148,Z 209.653,A -85,B 0,C 180,E1 -24506.222,E2 -24506.222} C_VEL
LIN {X 0,Y 143.354,Z 210.603,A -85,B 0,C 180,E1 -24509.357,E2 -24509.357} C_VEL
LIN {X 0,Y 143.679,Z 212.81,A -85,B 0,C 180,E1 -24514.727,E2 -24514.727} C_VEL
LIN {X 0,Y 144.662,Z 215.55,A -85,B 0,C 180,E1 -24515.58,E2 -24515.58} C_VEL
LIN {X 0,Y 146.978,Z 218.465,A -85,B 0,C 180,E1 -24517.122,E2 -24517.122} C_VEL
LIN {X 0,Y 149.015,Z 222.677,A -85,B 0,C 180,E1 -24518.675,E2 -24518.675} C_VEL
LIN {X 0,Y 150.327,Z 224.82,A -85,B 0,C 180,E1 -24519.567,E2 -24519.567} C_VEL
LIN {X 0,Y 152.971,Z 230.266,A -85,B 0,C 180,E1 -24521.552,E2 -24521.552} C_VEL
LIN {X 0,Y 156.11,Z 237.582,A -85,B 0,C 180,E1 -24524.071,E2 -24524.071} C_VEL
LIN {X 0,Y 158.481,Z 245.957,A -85,B 0,C 180,E1 -24526.611,E2 -24526.611} C_VEL
LIN {X 0,Y 159.253,Z 255.472,A -85,B 0,C 180,E1 -24529.143,E2 -24529.143} C_VEL
LIN {X 0,Y 159.167,Z 265.032,A -85,B 0,C 180,E1 -24531.823,E2 -24531.823} C_VEL
LIN {X 0,Y 158.325,Z 274.524,A -85,B 0,C 180,E1 -24534.761,E2 -24534.761} C_VEL
LIN {X 0,Y 157.08,Z 280.576,A -85,B 0,C 180,E1 -24536.769,E2 -24536.769} C_VEL
LIN {X 0,Y 152.753,Z 290.507,A -85,B 0,C 180,E1 -24540.361,E2 -24540.361} C_VEL
LIN {X 0,Y 149.66,Z 297.453,A -85,B 0,C 180,E1 -24543.623,E2 -24543.623} C_VEL
LIN {X 0,Y 146.512,Z 303.906,A -85,B 0,C 180,E1 -24547.438,E2 -24547.438} C_VEL
LIN {X 0,Y 143.941,Z 309.201,A -85,B 0,C 180,E1 -24551.5,E2 -24551.5} C_VEL
LIN {X 0,Y 142.181,Z 313.325,A -85,B 0,C 180,E1 -24555.694,E2 -24555.694} C_VEL
LIN {X 0,Y 141.396,Z 315.488,A -85,B 0,C 180,E1 -24558.535,E2 -24558.535} C_VEL
LIN {X 0,Y 140.849,Z 317.187,A -85,B 0,C 180,E1 -24561.393,E2 -24561.393} C_VEL
LIN {X 0,Y 140.553,Z 318.481,A -85,B 0,C 180,E1 -24564.263,E2 -24564.263} C_VEL
LIN {X 0,Y 140.568,Z 319.782,A -85,B 0,C 180,E1 -24569.358,E2 -24569.358} C_VEL
LIN {X 0,Y 140.504,Z 319.903,A -85,B 0,C 180,E1 -24572.869,E2 -24572.869} C_VEL
LIN {X 0,Y 140.853,Z 318.847,A -85,B 0,C 180,E1 -24578.61,E2 -24578.61} C_VEL
LIN {X 0,Y 141.417,Z 317.711,A -85,B 0,C 180,E1 -24581.467,E2 -24581.467} C_VEL
LIN {X 0,Y 142.254,Z 316.139,A -85,B 0,C 180,E1 -24584.302,E2 -24584.302} C_VEL
LIN {X 0,Y 144.072,Z 312.997,A -85,B 0,C 180,E1 -24588.487,E2 -24588.487} C_VEL
LIN {X 0,Y 146.731,Z 308.805,A -85,B 0,C 180,E1 -24592.531,E2 -24592.531} C_VEL
LIN {X 0,Y 150.677,Z 302.435,A -85,B 0,C 180,E1 -24597.05,E2 -24597.05} C_VEL
LIN {X 0,Y 154.512,Z 295.501,A -85,B 0,C 180,E1 -24600.777,E2 -24600.777} C_VEL
LIN {X 0,Y 159.169,Z 286.827,A -85,B 0,C 180,E1 -24604.26,E2 -24604.26} C_VEL
LIN {X 0,Y 160.732,Z 283.497,A -85,B 0,C 180,E1 -24605.404,E2 -24605.404} C_VEL
LIN {X 0,Y 162.264,Z 275.671,A -85,B 0,C 180,E1 -24608.221,E2 -24608.221} C_VEL
LIN {X 0,Y 163.15,Z 266.345,A -85,B 0,C 180,E1 -24611.273,E2 -24611.273} C_VEL
LIN {X 0,Y 163.2,Z 256.696,A -85,B 0,C 180,E1 -24614.213,E2 -24614.213} C_VEL
LIN {X 0,Y 162.292,Z 250.773,A -85,B 0,C 180,E1 -24616.143,E2 -24616.143} C_VEL
LIN {X 0,Y 160.072,Z 243.544,A -85,B 0,C 180,E1 -24618.809,E2 -24618.809} C_VEL
LIN {X 0,Y 156.736,Z 235.375,A -85,B 0,C 180,E1 -24622.148,E2 -24622.148} C_VEL
LIN {X 0,Y 153.792,Z 229.33,A -85,B 0,C 180,E1 -24624.885,E2 -24624.885} C_VEL
LIN {X 0,Y 153.126,Z 228.349,A -85,B 0,C 180,E1 -24625.436,E2 -24625.436} C_VEL
LIN {X 0,Y 148.499,Z 223.6,A -85,B 0,C 180,E1 -24629.174,E2 -24629.174} C_VEL
LIN {X 0,Y 143.871,Z 220.153,A -85,B 0,C 180,E1 -24633.25,E2 -24633.25} C_VEL
LIN {X 0,Y 140.993,Z 218.384,A -85,B 0,C 180,E1 -24636.14,E2 -24636.14} C_VEL
LIN {X 0,Y 138.186,Z 215.403,A -85,B 0,C 180,E1 -24639.729,E2 -24639.729} C_VEL
LIN {X 0,Y 136.619,Z 212.238,A -85,B 0,C 180,E1 -24642.506,E2 -24642.506} C_VEL
LIN {X 0,Y 136.459,Z 211.537,A -85,B 0,C 180,E1 -24642.968,E2 -24642.968} C_VEL
LIN {X 0,Y 136.426,Z 210.49,A -85,B 0,C 180,E1 -24648.167,E2 -24648.167} C_VEL
LIN {X 0,Y 136.543,Z 210.477,A -85,B 0,C 180,E1 -24651.118,E2 -24651.118} C_VEL
LIN {X 0,Y 137.121,Z 210.403,A -85,B 0,C 180,E1 -24660.001,E2 -24660.001} C_VEL
LIN {X 0,Y 136.499,Z 210.474,A -85,B 0,C 180,E1 -24666.965,E2 -24666.965} C_VEL
LIN {X 0,Y 136.41,Z 210.49,A -85,B 0,C 180,E1 -24671.894,E2 -24671.894} C_VEL
LIN {X 0,Y 136.253,Z 210.61,A -85,B 0,C 180,E1 -24675.138,E2 -24675.138} C_VEL
LIN {X 0,Y 136.869,Z 212.694,A -85,B 0,C 180,E1 -24676.597,E2 -24676.597} C_VEL
LIN {X 0,Y 138.821,Z 215.164,A -85,B 0,C 180,E1 -24679.598,E2 -24679.598} C_VEL
LIN {X 0,Y 140.707,Z 216.449,A -85,B 0,C 180,E1 -24681.895,E2 -24681.895} C_VEL
LIN {X 0,Y 142.073,Z 219.418,A -85,B 0,C 180,E1 -24683.893,E2 -24683.893} C_VEL
LIN {X 0,Y 144.545,Z 221.896,A -85,B 0,C 180,E1 -24686.534,E2 -24686.534} C_VEL
LIN {X 0,Y 146.382,Z 225.255,A -85,B 0,C 180,E1 -24688.694,E2 -24688.694} C_VEL
LIN {X 0,Y 147.694,Z 226.837,A -85,B 0,C 180,E1 -24689.977,E2 -24689.977} C_VEL
LIN {X 0,Y 150.117,Z 231.223,A -85,B 0,C 180,E1 -24692.577,E2 -24692.577} C_VEL
LIN {X 0,Y 153.989,Z 239.951,A -85,B 0,C 180,E1 -24696.999,E2 -24696.999} C_VEL
LIN {X 0,Y 156.517,Z 247.099,A -85,B 0,C 180,E1 -24700.243,E2 -24700.243} C_VEL
LIN {X 0,Y 158.073,Z 254.268,A -85,B 0,C 180,E1 -24703.163,E2 -24703.163} C_VEL
LIN {X 0,Y 158.587,Z 261.964,A -85,B 0,C 180,E1 -24706.068,E2 -24706.068} C_VEL
LIN {X 0,Y 158.327,Z 269.603,A -85,B 0,C 180,E1 -24708.993,E2 -24708.993} C_VEL
LIN {X 0,Y 157.998,Z 272.997,A -85,B 0,C 180,E1 -24710.352,E2 -24710.352} C_VEL
LIN {X 0,Y 156.148,Z 277.235,A -85,B 0,C 180,E1 -24711.768,E2 -24711.768} C_VEL
LIN {X 0,Y 151.14,Z 286.313,A -85,B 0,C 180,E1 -24715.277,E2 -24715.277} C_VEL
LIN {X 0,Y 146.615,Z 293.619,A -85,B 0,C 180,E1 -24718.983,E2 -24718.983} C_VEL
LIN {X 0,Y 142.964,Z 299.254,A -85,B 0,C 180,E1 -24722.768,E2 -24722.768} C_VEL
LIN {X 0,Y 140.212,Z 303.355,A -85,B 0,C 180,E1 -24726.359,E2 -24726.359} C_VEL
LIN {X 0,Y 137.483,Z 307.035,A -85,B 0,C 180,E1 -24730.593,E2 -24730.593} C_VEL
LIN {X 0,Y 135.613,Z 309.694,A -85,B 0,C 180,E1 -24734.981,E2 -24734.981} C_VEL
LIN {X 0,Y 134.711,Z 310.944,A -85,B 0,C 180,E1 -24737.954,E2 -24737.954} C_VEL
LIN {X 0,Y 134.055,Z 311.803,A -85,B 0,C 180,E1 -24740.95,E2 -24740.95} C_VEL
LIN {X 0,Y 133.655,Z 312.233,A -85,B 0,C 180,E1 -24743.962,E2 -24743.962} C_VEL
LIN {X 0,Y 133.544,Z 312.042,A -85,B 0,C 180,E1 -24749.32,E2 -24749.32} C_VEL
LIN {X 0,Y 133.949,Z 310.683,A -85,B 0,C 180,E1 -24754.51,E2 -24754.51} C_VEL
LIN {X 0,Y 134.936,Z 308.522,A -85,B 0,C 180,E1 -24758.987,E2 -24758.987} C_VEL
LIN {X 0,Y 136.384,Z 305.406,A -85,B 0,C 180,E1 -24763.405,E2 -24763.405} C_VEL
LIN {X 0,Y 138.523,Z 301.238,A -85,B 0,C 180,E1 -24767.719,E2 -24767.719} C_VEL
LIN {X 0,Y 141.898,Z 294.896,A -85,B 0,C 180,E1 -24772.568,E2 -24772.568} C_VEL
LIN {X 0,Y 145.594,Z 287.968,A -85,B 0,C 180,E1 -24776.516,E2 -24776.516} C_VEL
LIN {X 0,Y 149.727,Z 279.291,A -85,B 0,C 180,E1 -24780.3,E2 -24780.3} C_VEL
LIN {X 0,Y 153.642,Z 270.402,A -85,B 0,C 180,E1 -24783.288,E2 -24783.288} C_VEL
LIN {X 0,Y 154.269,Z 268.861,A -85,B 0,C 180,E1 -24783.752,E2 -24783.752} C_VEL
LIN {X 0,Y 154.798,Z 260.421,A -85,B 0,C 180,E1 -24786.704,E2 -24786.704} C_VEL
LIN {X 0,Y 154.326,Z 250.873,A -85,B 0,C 180,E1 -24789.88,E2 -24789.88} C_VEL
LIN {X 0,Y 152.883,Z 242.585,A -85,B 0,C 180,E1 -24792.648,E2 -24792.648} C_VEL
LIN {X 0,Y 149.62,Z 233.356,A -85,B 0,C 180,E1 -24796.143,E2 -24796.143} C_VEL
LIN {X 0,Y 147.448,Z 228.493,A -85,B 0,C 180,E1 -24798.14,E2 -24798.14} C_VEL
LIN {X 0,Y 145.039,Z 224.41,A -85,B 0,C 180,E1 -24800.111,E2 -24800.111} C_VEL
LIN {X 0,Y 143.062,Z 221.097,A -85,B 0,C 180,E1 -24801.755,E2 -24801.755} C_VEL
LIN {X 0,Y 140.411,Z 217.525,A -85,B 0,C 180,E1 -24803.864,E2 -24803.864} C_VEL
LIN {X 0,Y 139.624,Z 215.837,A -85,B 0,C 180,E1 -24804.629,E2 -24804.629} C_VEL
LIN {X 0,Y 137.413,Z 213.83,A -85,B 0,C 180,E1 -24806.354,E2 -24806.354} C_VEL
LIN {X 0,Y 136.184,Z 210.968,A -85,B 0,C 180,E1 -24807.627,E2 -24807.627} C_VEL
LIN {X 0,Y 136.108,Z 210.527,A -85,B 0,C 180,E1 -24807.825,E2 -24807.825} C_VEL
LIN {X 0,Y 136.134,Z 210.526,A -85,B 0,C 180,E1 -24812.313,E2 -24812.313} C_VEL
LIN {X 0,Y 136.265,Z 210.445,A -85,B 0,C 180,E1 -24818.836,E2 -24818.836} C_VEL
LIN {X 0,Y 136.28,Z 210.508,A -85,B 0,C 180,E1 -24825.057,E2 -24825.057} C_VEL
LIN {X 0,Y 136.488,Z 210.468,A -85,B 0,C 180,E1 -24828.113,E2 -24828.113} C_VEL
LIN {X 0,Y 136.593,Z 210.461,A -85,B 0,C 180,E1 -24831.12,E2 -24831.12} C_VEL
LIN {X 0,Y 137.113,Z 210.406,A -85,B 0,C 180,E1 -24839.999,E2 -24839.999} C_VEL
LIN {X 0,Y 136.573,Z 210.474,A -85,B 0,C 180,E1 -24848.88,E2 -24848.88} C_VEL
LIN {X 0,Y 136.478,Z 210.485,A -85,B 0,C 180,E1 -24851.955,E2 -24851.955} C_VEL
LIN {X 0,Y 136.247,Z 210.516,A -85,B 0,C 180,E1 -24858.028,E2 -24858.028} C_VEL
LIN {X 0,Y 136.214,Z 210.52,A -85,B 0,C 180,E1 -24861.78,E2 -24861.78} C_VEL
LIN {X 0,Y 136.084,Z 210.534,A -85,B 0,C 180,E1 -24864.403,E2 -24864.403} C_VEL
LIN {X 0,Y 136.426,Z 212.339,A -85,B 0,C 180,E1 -24870.023,E2 -24870.023} C_VEL
LIN {X 0,Y 136.506,Z 212.787,A -85,B 0,C 180,E1 -24870.331,E2 -24870.331} C_VEL
LIN {X 0,Y 137.904,Z 215.93,A -85,B 0,C 180,E1 -24871.705,E2 -24871.705} C_VEL
LIN {X 0,Y 140.284,Z 218.921,A -85,B 0,C 180,E1 -24873.589,E2 -24873.589} C_VEL
LIN {X 0,Y 142.141,Z 222.659,A -85,B 0,C 180,E1 -24875.247,E2 -24875.247} C_VEL
LIN {X 0,Y 143.428,Z 224.546,A -85,B 0,C 180,E1 -24876.232,E2 -24876.232} C_VEL
LIN {X 0,Y 145.401,Z 228.526,A -85,B 0,C 180,E1 -24877.934,E2 -24877.934} C_VEL
LIN {X 0,Y 148.547,Z 235.356,A -85,B 0,C 180,E1 -24880.672,E2 -24880.672} C_VEL
LIN {X 0,Y 151.526,Z 243.415,A -85,B 0,C 180,E1 -24883.624,E2 -24883.624} C_VEL
LIN {X 0,Y 152.908,Z 249.2,A -85,B 0,C 180,E1 -24885.52,E2 -24885.52} C_VEL
LIN {X 0,Y 153.352,Z 257.736,A -85,B 0,C 180,E1 -24887.968,E2 -24887.968} C_VEL
LIN {X 0,Y 152.92,Z 268.362,A -85,B 0,C 180,E1 -24891.21,E2 -24891.21} C_VEL
LIN {X 0,Y 151.882,Z 276.3,A -85,B 0,C 180,E1 -24893.85,E2 -24893.85} C_VEL
LIN {X 0,Y 151.016,Z 280.248,A -85,B 0,C 180,E1 -24895.248,E2 -24895.248} C_VEL
LIN {X 0,Y 147.297,Z 288.715,A -85,B 0,C 180,E1 -24898.347,E2 -24898.347} C_VEL
LIN {X 0,Y 143.604,Z 296.479,A -85,B 0,C 180,E1 -24901.976,E2 -24901.976} C_VEL
LIN {X 0,Y 139.924,Z 303.64,A -85,B 0,C 180,E1 -24906.312,E2 -24906.312} C_VEL
LIN {X 0,Y 137.2,Z 308.949,A -85,B 0,C 180,E1 -24910.555,E2 -24910.555} C_VEL
LIN {X 0,Y 135.287,Z 313.085,A -85,B 0,C 180,E1 -24914.948,E2 -24914.948} C_VEL
LIN {X 0,Y 134.426,Z 315.26,A -85,B 0,C 180,E1 -24917.932,E2 -24917.932} C_VEL
LIN {X 0,Y 133.822,Z 316.965,A -85,B 0,C 180,E1 -24920.938,E2 -24920.938} C_VEL
LIN {X 0,Y 133.396,Z 319.17,A -85,B 0,C 180,E1 -24926.982,E2 -24926.982} C_VEL
LIN {X 0,Y 133.531,Z 319.653,A -85,B 0,C 180,E1 -24930.002,E2 -24930.002} C_VEL
LIN {X 0,Y 133.406,Z 319.707,A -85,B 0,C 180,E1 -24933.022,E2 -24933.022} C_VEL
LIN {X 0,Y 133.827,Z 318.662,A -85,B 0,C 180,E1 -24939.066,E2 -24939.066} C_VEL
LIN {X 0,Y 134.452,Z 317.536,A -85,B 0,C 180,E1 -24942.07,E2 -24942.07} C_VEL
LIN {X 0,Y 135.358,Z 315.97,A -85,B 0,C 180,E1 -24945.048,E2 -24945.048} C_VEL
LIN {X 0,Y 137.328,Z 312.839,A -85,B 0,C 180,E1 -24949.43,E2 -24949.43} C_VEL
LIN {X 0,Y 140.153,Z 308.66,A -85,B 0,C 180,E1 -24953.651,E2 -24953.651} C_VEL
LIN {X 0,Y 144.336,Z 302.303,A -85,B 0,C 180,E1 -24958.343,E2 -24958.343} C_VEL
LIN {X 0,Y 148.422,Z 295.385,A -85,B 0,C 180,E1 -24962.188,E2 -24962.188} C_VEL
LIN {X 0,Y 153.344,Z 286.736,A -85,B 0,C 180,E1 -24965.757,E2 -24965.757} C_VEL
LIN {X 0,Y 154.752,Z 283.413,A -85,B 0,C 180,E1 -24966.994,E2 -24966.994} C_VEL
LIN {X 0,Y 156.18,Z 276.71,A -85,B 0,C 180,E1 -24969.535,E2 -24969.535} C_VEL
LIN {X 0,Y 157.336,Z 266.931,A -85,B 0,C 180,E1 -24972.94,E2 -24972.94} C_VEL
LIN {X 0,Y 157.508,Z 258.94,A -85,B 0,C 180,E1 -24975.553,E2 -24975.553} C_VEL
LIN {X 0,Y 156.598,Z 253.122,A -85,B 0,C 180,E1 -24977.687,E2 -24977.687} C_VEL
LIN {X 0,Y 154.422,Z 245.848,A -85,B 0,C 180,E1 -24980.685,E2 -24980.685} C_VEL
LIN {X 0,Y 151.721,Z 238.965,A -85,B 0,C 180,E1 -24983.801,E2 -24983.801} C_VEL
LIN {X 0,Y 149.336,Z 233.788,A -85,B 0,C 180,E1 -24986.405,E2 -24986.405} C_VEL
LIN {X 0,Y 147.156,Z 229.313,A -85,B 0,C 180,E1 -24988.831,E2 -24988.831} C_VEL
LIN {X 0,Y 145.106,Z 225.475,A -85,B 0,C 180,E1 -24991.131,E2 -24991.131} C_VEL
LIN {X 0,Y 144.468,Z 224.298,A -85,B 0,C 180,E1 -24991.884,E2 -24991.884} C_VEL
LIN {X 0,Y 141.869,Z 220.673,A -85,B 0,C 180,E1 -24994.804,E2 -24994.804} C_VEL
LIN {X 0,Y 140.993,Z 218.384,A -85,B 0,C 180,E1 -24996.14,E2 -24996.14} C_VEL
LIN {X 0,Y 138.276,Z 217.349,A -85,B 0,C 180,E1 -24999.178,E2 -24999.178} C_VEL
LIN {X 0,Y 132.862,Z 216.617,A -85,B 0,C 180,E1 -25007.297,E2 -25007.297} C_VEL
LIN {X 0,Y 132.178,Z 216.161,A -85,B 0,C 180,E1 -25008.984,E2 -25008.984} C_VEL
LIN {X 0,Y 130.605,Z 213.205,A -85,B 0,C 180,E1 -25020.001,E2 -25020.001} C_VEL
LIN {X 0,Y 134.265,Z 217.487,A -85,B 0,C 180,E1 -25034.301,E2 -25034.301} C_VEL
LIN {X 0,Y 135.49,Z 220.472,A -85,B 0,C 180,E1 -25037.159,E2 -25037.159} C_VEL
LIN {X 0,Y 138.109,Z 222.939,A -85,B 0,C 180,E1 -25041.064,E2 -25041.064} C_VEL
LIN {X 0,Y 139.525,Z 225.904,A -85,B 0,C 180,E1 -25043.371,E2 -25043.371} C_VEL
LIN {X 0,Y 140.894,Z 227.492,A -85,B 0,C 180,E1 -25045.088,E2 -25045.088} C_VEL
LIN {X 0,Y 144.16,Z 232.679,A -85,B 0,C 180,E1 -25049.178,E2 -25049.178} C_VEL
LIN {X 0,Y 147.293,Z 239.464,A -85,B 0,C 180,E1 -25053.281,E2 -25053.281} C_VEL
LIN {X 0,Y 150.082,Z 247.061,A -85,B 0,C 180,E1 -25057.246,E2 -25057.246} C_VEL
LIN {X 0,Y 151.904,Z 253.562,A -85,B 0,C 180,E1 -25060.371,E2 -25060.371} C_VEL
LIN {X 0,Y 152.721,Z 260.306,A -85,B 0,C 180,E1 -25063.224,E2 -25063.224} C_VEL
LIN {X 0,Y 152.578,Z 267.853,A -85,B 0,C 180,E1 -25066.298,E2 -25066.298} C_VEL
LIN {X 0,Y 151.892,Z 274.203,A -85,B 0,C 180,E1 -25068.969,E2 -25068.969} C_VEL
LIN {X 0,Y 151.498,Z 275.537,A -85,B 0,C 180,E1 -25069.5,E2 -25069.5} C_VEL
LIN {X 0,Y 147.01,Z 283.597,A -85,B 0,C 180,E1 -25072.445,E2 -25072.445} C_VEL
LIN {X 0,Y 142.046,Z 291.5,A -85,B 0,C 180,E1 -25076.178,E2 -25076.178} C_VEL
LIN {X 0,Y 137.763,Z 297.768,A -85,B 0,C 180,E1 -25080.143,E2 -25080.143} C_VEL
LIN {X 0,Y 133.715,Z 303.503,A -85,B 0,C 180,E1 -25085.135,E2 -25085.135} C_VEL
LIN {X 0,Y 130.794,Z 307.195,A -85,B 0,C 180,E1 -25089.557,E2 -25089.557} C_VEL
LIN {X 0,Y 128.726,Z 309.867,A -85,B 0,C 180,E1 -25094.157,E2 -25094.157} C_VEL
LIN {X 0,Y 127.038,Z 311.988,A -85,B 0,C 180,E1 -25100.445,E2 -25100.445} C_VEL
LIN {X 0,Y 126.586,Z 312.429,A -85,B 0,C 180,E1 -25103.623,E2 -25103.623} C_VEL
LIN {X 0,Y 126.453,Z 312.472,A -85,B 0,C 180,E1 -25106.812,E2 -25106.812} C_VEL
LIN {X 0,Y 126.476,Z 312.14,A -85,B 0,C 180,E1 -25109.998,E2 -25109.998} C_VEL
LIN {X 0,Y 126.701,Z 311.432,A -85,B 0,C 180,E1 -25113.177,E2 -25113.177} C_VEL
LIN {X 0,Y 127.171,Z 310.302,A -85,B 0,C 180,E1 -25116.343,E2 -25116.343} C_VEL
LIN {X 0,Y 127.934,Z 308.752,A -85,B 0,C 180,E1 -25119.483,E2 -25119.483} C_VEL
LIN {X 0,Y 129.499,Z 305.648,A -85,B 0,C 180,E1 -25124.132,E2 -25124.132} C_VEL
LIN {X 0,Y 131.795,Z 301.493,A -85,B 0,C 180,E1 -25128.656,E2 -25128.656} C_VEL
LIN {X 0,Y 135.385,Z 295.165,A -85,B 0,C 180,E1 -25133.719,E2 -25133.719} C_VEL
LIN {X 0,Y 139.305,Z 288.258,A -85,B 0,C 180,E1 -25137.814,E2 -25137.814} C_VEL
LIN {X 0,Y 143.666,Z 279.604,A -85,B 0,C 180,E1 -25141.723,E2 -25141.723} C_VEL
LIN {X 0,Y 147.772,Z 270.739,A -85,B 0,C 180,E1 -25144.795,E2 -25144.795} C_VEL
LIN {X 0,Y 148.386,Z 267.585,A -85,B 0,C 180,E1 -25145.943,E2 -25145.943} C_VEL
LIN {X 0,Y 148.684,Z 259.755,A -85,B 0,C 180,E1 -25148.869,E2 -25148.869} C_VEL
LIN {X 0,Y 148.39,Z 252.218,A -85,B 0,C 180,E1 -25151.528,E2 -25151.528} C_VEL
LIN {X 0,Y 147.095,Z 245.025,A -85,B 0,C 180,E1 -25154.218,E2 -25154.218} C_VEL
LIN {X 0,Y 144.78,Z 237.814,A -85,B 0,C 180,E1 -25157.187,E2 -25157.187} C_VEL
LIN {X 0,Y 141.531,Z 230.535,A -85,B 0,C 180,E1 -25160.594,E2 -25160.594} C_VEL
LIN {X 0,Y 138.211,Z 225.297,A -85,B 0,C 180,E1 -25163.649,E2 -25163.649} C_VEL
LIN {X 0,Y 136.083,Z 221.738,A -85,B 0,C 180,E1 -25165.744,E2 -25165.744} C_VEL
LIN {X 0,Y 133.956,Z 219.139,A -85,B 0,C 180,E1 -25167.745,E2 -25167.745} C_VEL
LIN {X 0,Y 132.991,Z 216.943,A -85,B 0,C 180,E1 -25168.903,E2 -25168.903} C_VEL
LIN {X 0,Y 130.632,Z 215.077,A -85,B 0,C 180,E1 -25171.179,E2 -25171.179} C_VEL
LIN {X 0,Y 129.251,Z 212.356,A -85,B 0,C 180,E1 -25172.909,E2 -25172.909} C_VEL
LIN {X 0,Y 129.037,Z 211.411,A -85,B 0,C 180,E1 -25173.407,E2 -25173.407} C_VEL
LIN {X 0,Y 129.117,Z 211.338,A -85,B 0,C 180,E1 -25177.702,E2 -25177.702} C_VEL
LIN {X 0,Y 129.172,Z 211.334,A -85,B 0,C 180,E1 -25180.946,E2 -25180.946} C_VEL
LIN {X 0,Y 129.406,Z 211.351,A -85,B 0,C 180,E1 -25187.814,E2 -25187.814} C_VEL
LIN {X 0,Y 129.516,Z 211.337,A -85,B 0,C 180,E1 -25190.63,E2 -25190.63} C_VEL
LIN {X 0,Y 130.07,Z 211.284,A -85,B 0,C 180,E1 -25199.999,E2 -25199.999} C_VEL
LIN {X 0,Y 129.5,Z 211.354,A -85,B 0,C 180,E1 -25209.369,E2 -25209.369} C_VEL
LIN {X 0,Y 129.38,Z 211.371,A -85,B 0,C 180,E1 -25212.549,E2 -25212.549} C_VEL
LIN {X 0,Y 129.163,Z 211.397,A -85,B 0,C 180,E1 -25219.054,E2 -25219.054} C_VEL
LIN {X 0,Y 129.123,Z 211.414,A -85,B 0,C 180,E1 -25222.395,E2 -25222.395} C_VEL
LIN {X 0,Y 129.149,Z 212.044,A -85,B 0,C 180,E1 -25224.408,E2 -25224.408} C_VEL
LIN {X 0,Y 130.166,Z 214.833,A -85,B 0,C 180,E1 -25225.805,E2 -25225.805} C_VEL
LIN {X 0,Y 133.039,Z 218.196,A -85,B 0,C 180,E1 -25228.697,E2 -25228.697} C_VEL
LIN {X 0,Y 133.74,Z 219.561,A -85,B 0,C 180,E1 -25229.461,E2 -25229.461} C_VEL
LIN {X 0,Y 135.545,Z 222.843,A -85,B 0,C 180,E1 -25231.34,E2 -25231.34} C_VEL
LIN {X 0,Y 136.751,Z 224.584,A -85,B 0,C 180,E1 -25232.439,E2 -25232.439} C_VEL
LIN {X 0,Y 138.788,Z 228.686,A -85,B 0,C 180,E1 -25234.507,E2 -25234.507} C_VEL
LIN {X 0,Y 143.298,Z 238.337,A -85,B 0,C 180,E1 -25238.999,E2 -25238.999} C_VEL
LIN {X 0,Y 146.139,Z 246.689,A -85,B 0,C 180,E1 -25242.32,E2 -25242.32} C_VEL
LIN {X 0,Y 147.408,Z 253.387,A -85,B 0,C 180,E1 -25244.687,E2 -25244.687} C_VEL
LIN {X 0,Y 147.367,Z 262.961,A -85,B 0,C 180,E1 -25247.68,E2 -25247.68} C_VEL
LIN {X 0,Y 146.254,Z 273.802,A -85,B 0,C 180,E1 -25251.346,E2 -25251.346} C_VEL
LIN {X 0,Y 145.013,Z 279.915,A -85,B 0,C 180,E1 -25253.586,E2 -25253.586} C_VEL
LIN {X 0,Y 142.848,Z 285.199,A -85,B 0,C 180,E1 -25255.548,E2 -25255.548} C_VEL
LIN {X 0,Y 138.389,Z 294.143,A -85,B 0,C 180,E1 -25259.484,E2 -25259.484} C_VEL
LIN {X 0,Y 134.604,Z 301.339,A -85,B 0,C 180,E1 -25263.657,E2 -25263.657} C_VEL
LIN {X 0,Y 131.417,Z 307.073,A -85,B 0,C 180,E1 -25268.02,E2 -25268.02} C_VEL
LIN {X 0,Y 128.967,Z 311.591,A -85,B 0,C 180,E1 -25272.563,E2 -25272.563} C_VEL
LIN {X 0,Y 127.452,Z 315.032,A -85,B 0,C 180,E1 -25277.261,E2 -25277.261} C_VEL
LIN {X 0,Y 126.79,Z 316.742,A -85,B 0,C 180,E1 -25280.431,E2 -25280.431} C_VEL
LIN {X 0,Y 126.41,Z 318.048,A -85,B 0,C 180,E1 -25283.619,E2 -25283.619} C_VEL
LIN {X 0,Y 126.302,Z 318.959,A -85,B 0,C 180,E1 -25286.813,E2 -25286.813} C_VEL
LIN {X 0,Y 126.427,Z 319.452,A -85,B 0,C 180,E1 -25290.002,E2 -25290.002} C_VEL
LIN {X 0,Y 126.308,Z 319.512,A -85,B 0,C 180,E1 -25293.192,E2 -25293.192} C_VEL
LIN {X 0,Y 126.797,Z 318.477,A -85,B 0,C 180,E1 -25299.573,E2 -25299.573} C_VEL
LIN {X 0,Y 127.481,Z 317.361,A -85,B 0,C 180,E1 -25302.741,E2 -25302.741} C_VEL
LIN {X 0,Y 128.476,Z 315.801,A -85,B 0,C 180,E1 -25305.875,E2 -25305.875} C_VEL
LIN {X 0,Y 130.63,Z 312.682,A -85,B 0,C 180,E1 -25310.47,E2 -25310.47} C_VEL
LIN {X 0,Y 133.638,Z 308.515,A -85,B 0,C 180,E1 -25314.88,E2 -25314.88} C_VEL
LIN {X 0,Y 138.079,Z 302.171,A -85,B 0,C 180,E1 -25319.753,E2 -25319.753} C_VEL
LIN {X 0,Y 142.457,Z 295.269,A -85,B 0,C 180,E1 -25323.711,E2 -25323.711} C_VEL
LIN {X 0,Y 147.613,Z 286.646,A -85,B 0,C 180,E1 -25327.375,E2 -25327.375} C_VEL
LIN {X 0,Y 148.877,Z 283.329,A -85,B 0,C 180,E1 -25328.717,E2 -25328.717} C_VEL
LIN {X 0,Y 150.671,Z 274.838,A -85,B 0,C 180,E1 -25332.081,E2 -25332.081} C_VEL
LIN {X 0,Y 151.75,Z 265.709,A -85,B 0,C 180,E1 -25335.38,E2 -25335.38} C_VEL
LIN {X 0,Y 151.754,Z 259.992,A -85,B 0,C 180,E1 -25337.448,E2 -25337.448} C_VEL
LIN {X 0,Y 150.322,Z 252.864,A -85,B 0,C 180,E1 -25340.477,E2 -25340.477} C_VEL
LIN {X 0,Y 147.753,Z 244.867,A -85,B 0,C 180,E1 -25344.278,E2 -25344.278} C_VEL
LIN {X 0,Y 145.595,Z 239.575,A -85,B 0,C 180,E1 -25347.109,E2 -25347.109} C_VEL
LIN {X 0,Y 143.74,Z 235.211,A -85,B 0,C 180,E1 -25349.602,E2 -25349.602} C_VEL
LIN {X 0,Y 140.879,Z 229.782,A -85,B 0,C 180,E1 -25353.322,E2 -25353.322} C_VEL
LIN {X 0,Y 138.711,Z 225.829,A -85,B 0,C 180,E1 -25356.386,E2 -25356.386} C_VEL
LIN {X 0,Y 138.132,Z 224.512,A -85,B 0,C 180,E1 -25357.371,E2 -25357.371} C_VEL
LIN {X 0,Y 135.317,Z 220.582,A -85,B 0,C 180,E1 -25361.843,E2 -25361.843} C_VEL
LIN {X 0,Y 134.381,Z 218.139,A -85,B 0,C 180,E1 -25364.064,E2 -25364.064} C_VEL
LIN {X 0,Y 132.178,Z 216.161,A -85,B 0,C 180,E1 -25368.984,E2 -25368.984} C_VEL
LIN {X 0,Y 131.297,Z 215.923,A -85,B 0,C 180,E1 -25371.523,E2 -25371.523} C_VEL
LIN {X 0,Y 130.485,Z 216.655,A -85,B 0,C 180,E1 -25374.078,E2 -25374.078} C_VEL
LIN {X 0,Y 129.114,Z 220.338,A -85,B 0,C 180,E1 -25380.954,E2 -25380.954} C_VEL
LIN {X 0,Y 129.116,Z 221.019,A -85,B 0,C 180,E1 -25382.714,E2 -25382.714} C_VEL
LIN {X 0,Y 132.067,Z 224.255,A -85,B 0,C 180,E1 -25393.66,E2 -25393.66} C_VEL
LIN {X 0,Y 133.25,Z 227.242,A -85,B 0,C 180,E1 -25396.864,E2 -25396.864} C_VEL
LIN {X 0,Y 135.069,Z 229.007,A -85,B 0,C 180,E1 -25399.927,E2 -25399.927} C_VEL
LIN {X 0,Y 136.545,Z 232.139,A -85,B 0,C 180,E1 -25402.708,E2 -25402.708} C_VEL
LIN {X 0,Y 137.521,Z 233.382,A -85,B 0,C 180,E1 -25404.133,E2 -25404.133} C_VEL
LIN {X 0,Y 140.288,Z 238.213,A -85,B 0,C 180,E1 -25408.22,E2 -25408.22} C_VEL
LIN {X 0,Y 142.652,Z 243.952,A -85,B 0,C 180,E1 -25411.981,E2 -25411.981} C_VEL
LIN {X 0,Y 144.789,Z 250.246,A -85,B 0,C 180,E1 -25415.626,E2 -25415.626} C_VEL
LIN {X 0,Y 146.557,Z 257.566,A -85,B 0,C 180,E1 -25419.45,E2 -25419.45} C_VEL
LIN {X 0,Y 146.989,Z 263.143,A -85,B 0,C 180,E1 -25422.021,E2 -25422.021} C_VEL
LIN {X 0,Y 146.526,Z 271.119,A -85,B 0,C 180,E1 -25425.538,E2 -25425.538} C_VEL
LIN {X 0,Y 145.829,Z 275.612,A -85,B 0,C 180,E1 -25427.57,E2 -25427.57} C_VEL
LIN {X 0,Y 145.206,Z 277.385,A -85,B 0,C 180,E1 -25428.28,E2 -25428.28} C_VEL
LIN {X 0,Y 139.652,Z 286.516,A -85,B 0,C 180,E1 -25431.941,E2 -25431.941} C_VEL
LIN {X 0,Y 134.578,Z 293.857,A -85,B 0,C 180,E1 -25435.848,E2 -25435.848} C_VEL
LIN {X 0,Y 129.631,Z 300.587,A -85,B 0,C 180,E1 -25440.795,E2 -25440.795} C_VEL
LIN {X 0,Y 126.163,Z 305.018,A -85,B 0,C 180,E1 -25445.304,E2 -25445.304} C_VEL
LIN {X 0,Y 123.264,Z 308.378,A -85,B 0,C 180,E1 -25449.995,E2 -25449.995} C_VEL
LIN {X 0,Y 120.802,Z 311.301,A -85,B 0,C 180,E1 -25456.542,E2 -25456.542} C_VEL
LIN {X 0,Y 120.023,Z 312.173,A -85,B 0,C 180,E1 -25459.881,E2 -25459.881} C_VEL
LIN {X 0,Y 119.541,Z 312.623,A -85,B 0,C 180,E1 -25463.246,E2 -25463.246} C_VEL
LIN {X 0,Y 119.366,Z 312.673,A -85,B 0,C 180,E1 -25466.623,E2 -25466.623} C_VEL
LIN {X 0,Y 119.395,Z 312.346,A -85,B 0,C 180,E1 -25469.998,E2 -25469.998} C_VEL
LIN {X 0,Y 119.627,Z 311.643,A -85,B 0,C 180,E1 -25473.366,E2 -25473.366} C_VEL
LIN {X 0,Y 120.147,Z 310.525,A -85,B 0,C 180,E1 -25476.716,E2 -25476.716} C_VEL
LIN {X 0,Y 120.936,Z 308.981,A -85,B 0,C 180,E1 -25480.037,E2 -25480.037} C_VEL
LIN {X 0,Y 122.634,Z 305.889,A -85,B 0,C 180,E1 -25484.941,E2 -25484.941} C_VEL
LIN {X 0,Y 125.09,Z 301.748,A -85,B 0,C 180,E1 -25489.697,E2 -25489.697} C_VEL
LIN {X 0,Y 128.936,Z 295.434,A -85,B 0,C 180,E1 -25494.984,E2 -25494.984} C_VEL
LIN {X 0,Y 133.072,Z 288.547,A -85,B 0,C 180,E1 -25499.239,E2 -25499.239} C_VEL
LIN {X 0,Y 137.68,Z 279.918,A -85,B 0,C 180,E1 -25503.276,E2 -25503.276} C_VEL
LIN {X 0,Y 141.974,Z 271.077,A -85,B 0,C 180,E1 -25506.438,E2 -25506.438} C_VEL
LIN {X 0,Y 142.652,Z 264.605,A -85,B 0,C 180,E1 -25509.066,E2 -25509.066} C_VEL
LIN {X 0,Y 142.741,Z 255.997,A -85,B 0,C 180,E1 -25512.392,E2 -25512.392} C_VEL
LIN {X 0,Y 141.863,Z 249.265,A -85,B 0,C 180,E1 -25515.086,E2 -25515.086} C_VEL
LIN {X 0,Y 139.879,Z 242.204,A -85,B 0,C 180,E1 -25518.261,E2 -25518.261} C_VEL
LIN {X 0,Y 137.574,Z 236.461,A -85,B 0,C 180,E1 -25521.165,E2 -25521.165} C_VEL
LIN {X 0,Y 134.198,Z 230.544,A -85,B 0,C 180,E1 -25524.824,E2 -25524.824} C_VEL
LIN {X 0,Y 133.119,Z 228.449,A -85,B 0,C 180,E1 -25526.093,E2 -25526.093} C_VEL
LIN {X 0,Y 130.346,Z 224.227,A -85,B 0,C 180,E1 -25529.243,E2 -25529.243} C_VEL
LIN {X 0,Y 129.751,Z 223.072,A -85,B 0,C 180,E1 -25530.021,E2 -25530.021} C_VEL
LIN {X 0,Y 127.583,Z 220.779,A -85,B 0,C 180,E1 -25532.525,E2 -25532.525} C_VEL
LIN {X 0,Y 126.327,Z 217.944,A -85,B 0,C 180,E1 -25534.458,E2 -25534.458} C_VEL
LIN {X 0,Y 123.978,Z 216.207,A -85,B 0,C 180,E1 -25537.532,E2 -25537.532} C_VEL
LIN {X 0,Y 122.59,Z 214.117,A -85,B 0,C 180,E1 -25539.88,E2 -25539.88} C_VEL
LIN {X 0,Y 122.143,Z 212.208,A -85,B 0,C 180,E1 -25541.115,E2 -25541.115} C_VEL
LIN {X 0,Y 122.353,Z 212.231,A -85,B 0,C 180,E1 -25547.521,E2 -25547.521} C_VEL
LIN {X 0,Y 122.443,Z 212.215,A -85,B 0,C 180,E1 -25550.084,E2 -25550.084} C_VEL
LIN {X 0,Y 122.588,Z 212.195,A -85,B 0,C 180,E1 -25556.713,E2 -25556.713} C_VEL
LIN {X 0,Y 123.024,Z 212.162,A -85,B 0,C 180,E1 -25559.999,E2 -25559.999} C_VEL
LIN {X 0,Y 122.432,Z 212.233,A -85,B 0,C 180,E1 -25566.592,E2 -25566.592} C_VEL
LIN {X 0,Y 122.43,Z 212.235,A -85,B 0,C 180,E1 -25569.916,E2 -25569.916} C_VEL
LIN {X 0,Y 122.156,Z 212.271,A -85,B 0,C 180,E1 -25575.859,E2 -25575.859} C_VEL
LIN {X 0,Y 122.137,Z 212.298,A -85,B 0,C 180,E1 -25576.398,E2 -25576.398} C_VEL
LIN {X 0,Y 122.672,Z 214.329,A -85,B 0,C 180,E1 -25577.719,E2 -25577.719} C_VEL
LIN {X 0,Y 124.707,Z 216.985,A -85,B 0,C 180,E1 -25580.901,E2 -25580.901} C_VEL
LIN {X 0,Y 126.561,Z 218.467,A -85,B 0,C 180,E1 -25583.198,E2 -25583.198} C_VEL
LIN {X 0,Y 128.018,Z 221.832,A -85,B 0,C 180,E1 -25585.397,E2 -25585.397} C_VEL
LIN {X 0,Y 130.274,Z 224.705,A -85,B 0,C 180,E1 -25587.947,E2 -25587.947} C_VEL
LIN {X 0,Y 132.097,Z 228.543,A -85,B 0,C 180,E1 -25590.249,E2 -25590.249} C_VEL
LIN {X 0,Y 132.887,Z 229.589,A -85,B 0,C 180,E1 -25591.04,E2 -25591.04} C_VEL
LIN {X 0,Y 136.483,Z 237.848,A -85,B 0,C 180,E1 -25595.401,E2 -25595.401} C_VEL
LIN {X 0,Y 139.02,Z 244.411,A -85,B 0,C 180,E1 -25598.546,E2 -25598.546} C_VEL
LIN {X 0,Y 141.14,Z 251.721,A -85,B 0,C 180,E1 -25601.684,E2 -25601.684} C_VEL
LIN {X 0,Y 141.767,Z 255.999,A -85,B 0,C 180,E1 -25603.318,E2 -25603.318} C_VEL
LIN {X 0,Y 141.436,Z 265.099,A -85,B 0,C 180,E1 -25606.403,E2 -25606.403} C_VEL
LIN {X 0,Y 139.997,Z 275.602,A -85,B 0,C 180,E1 -25610.209,E2 -25610.209} C_VEL
LIN {X 0,Y 138.569,Z 281.405,A -85,B 0,C 180,E1 -25612.516,E2 -25612.516} C_VEL
LIN {X 0,Y 135.352,Z 288.12,A -85,B 0,C 180,E1 -25615.174,E2 -25615.174} C_VEL
LIN {X 0,Y 131.022,Z 296.072,A -85,B 0,C 180,E1 -25619.119,E2 -25619.119} C_VEL
LIN {X 0,Y 127.608,Z 302.095,A -85,B 0,C 180,E1 -25622.98,E2 -25622.98} C_VEL
LIN {X 0,Y 123.861,Z 308.446,A -85,B 0,C 180,E1 -25628.361,E2 -25628.361} C_VEL
LIN {X 0,Y 121.533,Z 312.604,A -85,B 0,C 180,E1 -25633.197,E2 -25633.197} C_VEL
LIN {X 0,Y 120.508,Z 314.803,A -85,B 0,C 180,E1 -25636.513,E2 -25636.513} C_VEL
LIN {X 0,Y 119.782,Z 316.52,A -85,B 0,C 180,E1 -25639.865,E2 -25639.865} C_VEL
LIN {X 0,Y 119.218,Z 318.748,A -85,B 0,C 180,E1 -25646.623,E2 -25646.623} C_VEL
LIN {X 0,Y 119.332,Z 319.252,A -85,B 0,C 180,E1 -25650.002,E2 -25650.002} C_VEL
LIN {X 0,Y 119.222,Z 319.317,A -85,B 0,C 180,E1 -25653.382,E2 -25653.382} C_VEL
LIN {X 0,Y 119.79,Z 318.292,A -85,B 0,C 180,E1 -25660.139,E2 -25660.139} C_VEL
LIN {X 0,Y 120.54,Z 317.186,A -85,B 0,C 180,E1 -25663.488,E2 -25663.488} C_VEL
LIN {X 0,Y 121.631,Z 315.632,A -85,B 0,C 180,E1 -25666.794,E2 -25666.794} C_VEL
LIN {X 0,Y 123.983,Z 312.525,A -85,B 0,C 180,E1 -25671.621,E2 -25671.621} C_VEL
LIN {X 0,Y 127.196,Z 308.369,A -85,B 0,C 180,E1 -25676.234,E2 -25676.234} C_VEL
LIN {X 0,Y 131.234,Z 303.051,A -85,B 0,C 180,E1 -25680.581,E2 -25680.581} C_VEL
LIN {X 0,Y 135.744,Z 296.388,A -85,B 0,C 180,E1 -25684.716,E2 -25684.716} C_VEL
LIN {X 0,Y 141.08,Z 288.132,A -85,B 0,C 180,E1 -25688.512,E2 -25688.512} C_VEL
LIN {X 0,Y 142.597,Z 284.92,A -85,B 0,C 180,E1 -25689.844,E2 -25689.844} C_VEL
LIN {X 0,Y 144.591,Z 277.071,A -85,B 0,C 180,E1 -25693.19,E2 -25693.19} C_VEL
LIN {X 0,Y 146.002,Z 268.04,A -85,B 0,C 180,E1 -25696.718,E2 -25696.718} C_VEL
LIN {X 0,Y 146.197,Z 263.185,A -85,B 0,C 180,E1 -25698.626,E2 -25698.626} C_VEL
LIN {X 0,Y 145.364,Z 257.916,A -85,B 0,C 180,E1 -25701.06,E2 -25701.06} C_VEL
LIN {X 0,Y 143.413,Z 250.474,A -85,B 0,C 180,E1 -25704.844,E2 -25704.844} C_VEL
LIN {X 0,Y 141.26,Z 244.347,A -85,B 0,C 180,E1 -25708.34,E2 -25708.34} C_VEL
LIN {X 0,Y 140.316,Z 241.646,A -85,B 0,C 180,E1 -25709.943,E2 -25709.943} C_VEL
LIN {X 0,Y 137.349,Z 235.292,A -85,B 0,C 180,E1 -25714.568,E2 -25714.568} C_VEL
LIN {X 0,Y 135.033,Z 230.486,A -85,B 0,C 180,E1 -25718.634,E2 -25718.634} C_VEL
LIN {X 0,Y 132.576,Z 225.996,A -85,B 0,C 180,E1 -25723.644,E2 -25723.644} C_VEL
LIN {X 0,Y 132.129,Z 224.706,A -85,B 0,C 180,E1 -25724.972,E2 -25724.972} C_VEL
LIN {X 0,Y 129.842,Z 222.322,A -85,B 0,C 180,E1 -25731.44,E2 -25731.44} C_VEL
LIN {X 0,Y 129.096,Z 220.23,A -85,B 0,C 180,E1 -25740.001,E2 -25740.001} C_VEL
LIN {X 0,Y 129.116,Z 221.019,A -85,B 0,C 180,E1 -25742.714,E2 -25742.714} C_VEL
LIN {X 0,Y 129.219,Z 222.444,A -85,B 0,C 180,E1 -25745.261,E2 -25745.261} C_VEL
LIN {X 0,Y 129.246,Z 226.596,A -85,B 0,C 180,E1 -25749.262,E2 -25749.262} C_VEL
LIN {X 0,Y 129.764,Z 231.914,A -85,B 0,C 180,E1 -25754.035,E2 -25754.035} C_VEL
LIN {X 0,Y 130.303,Z 233.174,A -85,B 0,C 180,E1 -25755.69,E2 -25755.69} C_VEL
LIN {X 0,Y 131.7,Z 235.04,A -85,B 0,C 180,E1 -25758.675,E2 -25758.675} C_VEL
LIN {X 0,Y 134.75,Z 240.709,A -85,B 0,C 180,E1 -25764.662,E2 -25764.662} C_VEL
LIN {X 0,Y 136.806,Z 245.143,A -85,B 0,C 180,E1 -25768.373,E2 -25768.373} C_VEL
LIN {X 0,Y 138.343,Z 249.452,A -85,B 0,C 180,E1 -25771.381,E2 -25771.381} C_VEL
LIN {X 0,Y 139.905,Z 255.088,A -85,B 0,C 180,E1 -25774.872,E2 -25774.872} C_VEL
LIN {X 0,Y 141.148,Z 261.48,A -85,B 0,C 180,E1 -25778.491,E2 -25778.491} C_VEL
LIN {X 0,Y 141.234,Z 267.083,A -85,B 0,C 180,E1 -25781.278,E2 -25781.278} C_VEL
LIN {X 0,Y 140.355,Z 274.7,A -85,B 0,C 180,E1 -25784.926,E2 -25784.926} C_VEL
LIN {X 0,Y 139.786,Z 277.461,A -85,B 0,C 180,E1 -25786.268,E2 -25786.268} C_VEL
LIN {X 0,Y 135.981,Z 283.782,A -85,B 0,C 180,E1 -25788.78,E2 -25788.78} C_VEL
LIN {X 0,Y 130.459,Z 291.725,A -85,B 0,C 180,E1 -25792.696,E2 -25792.696} C_VEL
LIN {X 0,Y 126.341,Z 297.089,A -85,B 0,C 180,E1 -25796.202,E2 -25796.202} C_VEL
LIN {X 0,Y 122.115,Z 302.332,A -85,B 0,C 180,E1 -25800.712,E2 -25800.712} C_VEL
LIN {X 0,Y 118.617,Z 306.406,A -85,B 0,C 180,E1 -25805.496,E2 -25805.496} C_VEL
LIN {X 0,Y 116.585,Z 308.545,A -85,B 0,C 180,E1 -25808.795,E2 -25808.795} C_VEL
LIN {X 0,Y 113.894,Z 311.479,A -85,B 0,C 180,E1 -25815.709,E2 -25815.709} C_VEL
LIN {X 0,Y 113.035,Z 312.357,A -85,B 0,C 180,E1 -25819.248,E2 -25819.248} C_VEL
LIN {X 0,Y 112.486,Z 312.818,A -85,B 0,C 180,E1 -25822.82,E2 -25822.82} C_VEL
LIN {X 0,Y 112.276,Z 312.873,A -85,B 0,C 180,E1 -25826.409,E2 -25826.409} C_VEL
LIN {X 0,Y 112.306,Z 312.552,A -85,B 0,C 180,E1 -25829.998,E2 -25829.998} C_VEL
LIN {X 0,Y 112.556,Z 311.855,A -85,B 0,C 180,E1 -25833.577,E2 -25833.577} C_VEL
LIN {X 0,Y 113.124,Z 310.748,A -85,B 0,C 180,E1 -25837.135,E2 -25837.135} C_VEL
LIN {X 0,Y 113.958,Z 309.211,A -85,B 0,C 180,E1 -25840.659,E2 -25840.659} C_VEL
LIN {X 0,Y 115.79,Z 306.131,A -85,B 0,C 180,E1 -25845.847,E2 -25845.847} C_VEL
LIN {X 0,Y 118.438,Z 302.003,A -85,B 0,C 180,E1 -25850.853,E2 -25850.853} C_VEL
LIN {X 0,Y 122.556,Z 295.703,A -85,B 0,C 180,E1 -25856.382,E2 -25856.382} C_VEL
LIN {X 0,Y 126.931,Z 288.835,A -85,B 0,C 180,E1 -25860.803,E2 -25860.803} C_VEL
LIN {X 0,Y 131.808,Z 280.231,A -85,B 0,C 180,E1 -25864.968,E2 -25864.968} C_VEL
LIN {X 0,Y 135.436,Z 273.351,A -85,B 0,C 180,E1 -25867.564,E2 -25867.564} C_VEL
LIN {X 0,Y 136.227,Z 270.22,A -85,B 0,C 180,E1 -25868.846,E2 -25868.846} C_VEL
LIN {X 0,Y 136.97,Z 261.439,A -85,B 0,C 180,E1 -25872.566,E2 -25872.566} C_VEL
LIN {X 0,Y 136.672,Z 254.173,A -85,B 0,C 180,E1 -25875.64,E2 -25875.64} C_VEL
LIN {X 0,Y 135.103,Z 247.206,A -85,B 0,C 180,E1 -25879.016,E2 -25879.016} C_VEL
LIN {X 0,Y 133.36,Z 242.068,A -85,B 0,C 180,E1 -25881.781,E2 -25881.781} C_VEL
LIN {X 0,Y 130.453,Z 236.338,A -85,B 0,C 180,E1 -25885.55,E2 -25885.55} C_VEL
LIN {X 0,Y 129.328,Z 234.051,A -85,B 0,C 180,E1 -25887.082,E2 -25887.082} C_VEL
LIN {X 0,Y 126.509,Z 229.19,A -85,B 0,C 180,E1 -25890.931,E2 -25890.931} C_VEL
LIN {X 0,Y 124.255,Z 226.171,A -85,B 0,C 180,E1 -25894.091,E2 -25894.091} C_VEL
LIN {X 0,Y 123.543,Z 224.41,A -85,B 0,C 180,E1 -25895.419,E2 -25895.419} C_VEL
LIN {X 0,Y 120.929,Z 221.778,A -85,B 0,C 180,E1 -25899.591,E2 -25899.591} C_VEL
LIN {X 0,Y 119.95,Z 219.058,A -85,B 0,C 180,E1 -25902.084,E2 -25902.084} C_VEL
LIN {X 0,Y 116.973,Z 216.782,A -85,B 0,C 180,E1 -25909.615,E2 -25909.615} C_VEL
LIN {X 0,Y 116.119,Z 213.817,A -85,B 0,C 180,E1 -25919.999,E2 -25919.999} C_VEL
LIN {X 0,Y 117.082,Z 216.956,A -85,B 0,C 180,E1 -25928.195,E2 -25928.195} C_VEL
LIN {X 0,Y 120.032,Z 219.211,A -85,B 0,C 180,E1 -25935.385,E2 -25935.385} C_VEL
LIN {X 0,Y 121.116,Z 221.889,A -85,B 0,C 180,E1 -25937.954,E2 -25937.954} C_VEL
LIN {X 0,Y 123.269,Z 224.139,A -85,B 0,C 180,E1 -25941.312,E2 -25941.312} C_VEL
LIN {X 0,Y 123.795,Z 224.761,A -85,B 0,C 180,E1 -25942.092,E2 -25942.092} C_VEL
LIN {X 0,Y 125.415,Z 228.43,A -85,B 0,C 180,E1 -25944.852,E2 -25944.852} C_VEL
LIN {X 0,Y 126.596,Z 229.97,A -85,B 0,C 180,E1 -25946.366,E2 -25946.366} C_VEL
LIN {X 0,Y 129.282,Z 235.569,A -85,B 0,C 180,E1 -25950.188,E2 -25950.188} C_VEL
LIN {X 0,Y 132.592,Z 244.032,A -85,B 0,C 180,E1 -25955.016,E2 -25955.016} C_VEL
LIN {X 0,Y 134.882,Z 251.428,A -85,B 0,C 180,E1 -25958.701,E2 -25958.701} C_VEL
LIN {X 0,Y 135.996,Z 257.014,A -85,B 0,C 180,E1 -25961.215,E2 -25961.215} C_VEL
LIN {X 0,Y 136.058,Z 261.527,A -85,B 0,C 180,E1 -25962.935,E2 -25962.935} C_VEL
LIN {X 0,Y 135.006,Z 270.875,A -85,B 0,C 180,E1 -25966.398,E2 -25966.398} C_VEL
LIN {X 0,Y 133.313,Z 279.236,A -85,B 0,C 180,E1 -25969.781,E2 -25969.781} C_VEL
LIN {X 0,Y 132.15,Z 282.883,A -85,B 0,C 180,E1 -25971.332,E2 -25971.332} C_VEL
LIN {X 0,Y 127.867,Z 290.809,A -85,B 0,C 180,E1 -25974.758,E2 -25974.758} C_VEL
LIN {X 0,Y 123.374,Z 298.553,A -85,B 0,C 180,E1 -25979.162,E2 -25979.162} C_VEL
LIN {X 0,Y 119.419,Z 304.763,A -85,B 0,C 180,E1 -25983.812,E2 -25983.812} C_VEL
LIN {X 0,Y 116.276,Z 309.699,A -85,B 0,C 180,E1 -25988.741,E2 -25988.741} C_VEL
LIN {X 0,Y 114.098,Z 313.51,A -85,B 0,C 180,E1 -25993.912,E2 -25993.912} C_VEL
LIN {X 0,Y 112.772,Z 316.297,A -85,B 0,C 180,E1 -25999.228,E2 -25999.228} C_VEL
LIN {X 0,Y 112.126,Z 318.537,A -85,B 0,C 180,E1 -26006.409,E2 -26006.409} C_VEL
LIN {X 0,Y 112.249,Z 319.051,A -85,B 0,C 180,E1 -26010.002,E2 -26010.002} C_VEL
LIN {X 0,Y 112.128,Z 319.121,A -85,B 0,C 180,E1 -26013.596,E2 -26013.596} C_VEL
LIN {X 0,Y 112.782,Z 318.107,A -85,B 0,C 180,E1 -26020.776,E2 -26020.776} C_VEL
LIN {X 0,Y 113.63,Z 317.01,A -85,B 0,C 180,E1 -26024.325,E2 -26024.325} C_VEL
LIN {X 0,Y 114.806,Z 315.463,A -85,B 0,C 180,E1 -26027.824,E2 -26027.824} C_VEL
LIN {X 0,Y 117.396,Z 312.368,A -85,B 0,C 180,E1 -26032.901,E2 -26032.901} C_VEL
LIN {X 0,Y 120.839,Z 308.224,A -85,B 0,C 180,E1 -26037.729,E2 -26037.729} C_VEL
LIN {X 0,Y 125.58,Z 302.303,A -85,B 0,C 180,E1 -26042.696,E2 -26042.696} C_VEL
LIN {X 0,Y 130.842,Z 295.037,A -85,B 0,C 180,E1 -26047.176,E2 -26047.176} C_VEL
LIN {X 0,Y 135.563,Z 288.033,A -85,B 0,C 180,E1 -26050.393,E2 -26050.393} C_VEL
LIN {X 0,Y 136.931,Z 284.826,A -85,B 0,C 180,E1 -26051.852,E2 -26051.852} C_VEL
LIN {X 0,Y 138.899,Z 277.636,A -85,B 0,C 180,E1 -26055.101,E2 -26055.101} C_VEL
LIN {X 0,Y 140.478,Z 269.161,A -85,B 0,C 180,E1 -26058.627,E2 -26058.627} C_VEL
LIN {X 0,Y 140.579,Z 265.596,A -85,B 0,C 180,E1 -26060.229,E2 -26060.229} C_VEL
LIN {X 0,Y 139.517,Z 258.912,A -85,B 0,C 180,E1 -26063.703,E2 -26063.703} C_VEL
LIN {X 0,Y 137.554,Z 251.117,A -85,B 0,C 180,E1 -26068.234,E2 -26068.234} C_VEL
LIN {X 0,Y 135.863,Z 246.113,A -85,B 0,C 180,E1 -26071.565,E2 -26071.565} C_VEL
LIN {X 0,Y 133.988,Z 241.391,A -85,B 0,C 180,E1 -26075.19,E2 -26075.19} C_VEL
LIN {X 0,Y 131.854,Z 236.405,A -85,B 0,C 180,E1 -26079.73,E2 -26079.73} C_VEL
LIN {X 0,Y 130.01,Z 232.519,A -85,B 0,C 180,E1 -26084.319,E2 -26084.319} C_VEL
LIN {X 0,Y 128.99,Z 230.551,A -85,B 0,C 180,E1 -26087.413,E2 -26087.413} C_VEL
LIN {X 0,Y 127.145,Z 227.828,A -85,B 0,C 180,E1 -26096.832,E2 -26096.832} C_VEL
LIN {X 0,Y 127.207,Z 227.16,A -85,B 0,C 180,E1 -26100.001,E2 -26100.001} C_VEL
LIN {X 0,Y 129.41,Z 230.553,A -85,B 0,C 180,E1 -26112.547,E2 -26112.547} C_VEL
LIN {X 0,Y 130.303,Z 233.174,A -85,B 0,C 180,E1 -26115.69,E2 -26115.69} C_VEL
LIN {X 0,Y 131.106,Z 235.36,A -85,B 0,C 180,E1 -26118.068,E2 -26118.068} C_VEL
LIN {X 0,Y 131.538,Z 238.477,A -85,B 0,C 180,E1 -26120.269,E2 -26120.269} C_VEL
LIN {X 0,Y 132.067,Z 248.122,A -85,B 0,C 180,E1 -26125.886,E2 -26125.886} C_VEL
LIN {X 0,Y 132.5,Z 250.208,A -85,B 0,C 180,E1 -26127.373,E2 -26127.373} C_VEL
LIN {X 0,Y 134.119,Z 255.981,A -85,B 0,C 180,E1 -26131.603,E2 -26131.603} C_VEL
LIN {X 0,Y 135.394,Z 262.882,A -85,B 0,C 180,E1 -26136.058,E2 -26136.058} C_VEL
LIN {X 0,Y 135.663,Z 268.014,A -85,B 0,C 180,E1 -26139.009,E2 -26139.009} C_VEL
LIN {X 0,Y 134.613,Z 275.771,A -85,B 0,C 180,E1 -26143.037,E2 -26143.037} C_VEL
LIN {X 0,Y 133.752,Z 279.197,A -85,B 0,C 180,E1 -26144.818,E2 -26144.818} C_VEL
LIN {X 0,Y 127.762,Z 288.071,A -85,B 0,C 180,E1 -26148.693,E2 -26148.693} C_VEL
LIN {X 0,Y 122.174,Z 295.201,A -85,B 0,C 180,E1 -26152.843,E2 -26152.843} C_VEL
LIN {X 0,Y 117.385,Z 300.87,A -85,B 0,C 180,E1 -26157.395,E2 -26157.395} C_VEL
LIN {X 0,Y 113.36,Z 305.326,A -85,B 0,C 180,E1 -26162.291,E2 -26162.291} C_VEL
LIN {X 0,Y 109.964,Z 308.711,A -85,B 0,C 180,E1 -26167.45,E2 -26167.45} C_VEL
LIN {X 0,Y 108.312,Z 310.385,A -85,B 0,C 180,E1 -26171.067,E2 -26171.067} C_VEL
LIN {X 0,Y 106.047,Z 312.541,A -85,B 0,C 180,E1 -26178.53,E2 -26178.53} C_VEL
LIN {X 0,Y 105.456,Z 313.013,A -85,B 0,C 180,E1 -26182.338,E2 -26182.338} C_VEL
LIN {X 0,Y 105.196,Z 313.074,A -85,B 0,C 180,E1 -26186.167,E2 -26186.167} C_VEL
LIN {X 0,Y 105.225,Z 312.758,A -85,B 0,C 180,E1 -26189.997,E2 -26189.997} C_VEL
LIN {X 0,Y 105.502,Z 312.066,A -85,B 0,C 180,E1 -26193.817,E2 -26193.817} C_VEL
LIN {X 0,Y 106.104,Z 310.97,A -85,B 0,C 180,E1 -26197.609,E2 -26197.609} C_VEL
LIN {X 0,Y 106.987,Z 309.44,A -85,B 0,C 180,E1 -26201.362,E2 -26201.362} C_VEL
LIN {X 0,Y 108.993,Z 306.373,A -85,B 0,C 180,E1 -26206.864,E2 -26206.864} C_VEL
LIN {X 0,Y 111.847,Z 302.257,A -85,B 0,C 180,E1 -26212.145,E2 -26212.145} C_VEL
LIN {X 0,Y 116.257,Z 295.971,A -85,B 0,C 180,E1 -26217.932,E2 -26217.932} C_VEL
LIN {X 0,Y 120.897,Z 289.121,A -85,B 0,C 180,E1 -26222.523,E2 -26222.523} C_VEL
LIN {X 0,Y 126.068,Z 280.543,A -85,B 0,C 180,E1 -26226.813,E2 -26226.813} C_VEL
LIN {X 0,Y 129.799,Z 273.69,A -85,B 0,C 180,E1 -26229.503,E2 -26229.503} C_VEL
LIN {X 0,Y 130.898,Z 266.797,A -85,B 0,C 180,E1 -26232.667,E2 -26232.667} C_VEL
LIN {X 0,Y 131.235,Z 259.739,A -85,B 0,C 180,E1 -26235.877,E2 -26235.877} C_VEL
LIN {X 0,Y 130.684,Z 254.691,A -85,B 0,C 180,E1 -26238.383,E2 -26238.383} C_VEL
LIN {X 0,Y 128.904,Z 247.452,A -85,B 0,C 180,E1 -26242.438,E2 -26242.438} C_VEL
LIN {X 0,Y 126.253,Z 241.568,A -85,B 0,C 180,E1 -26246.604,E2 -26246.604} C_VEL
LIN {X 0,Y 123.49,Z 236.065,A -85,B 0,C 180,E1 -26251.068,E2 -26251.068} C_VEL
LIN {X 0,Y 121.501,Z 232.994,A -85,B 0,C 180,E1 -26254.288,E2 -26254.288} C_VEL
LIN {X 0,Y 120.731,Z 231.111,A -85,B 0,C 180,E1 -26255.952,E2 -26255.952} C_VEL
LIN {X 0,Y 118.167,Z 227.759,A -85,B 0,C 180,E1 -26260.905,E2 -26260.905} C_VEL
LIN {X 0,Y 117.486,Z 225.623,A -85,B 0,C 180,E1 -26263.139,E2 -26263.139} C_VEL
LIN {X 0,Y 114.556,Z 220.971,A -85,B 0,C 180,E1 -26279.999,E2 -26279.999} C_VEL
LIN {X 0,Y 116.354,Z 224.841,A -85,B 0,C 180,E1 -26291.32,E2 -26291.32} C_VEL
LIN {X 0,Y 117.706,Z 225.838,A -85,B 0,C 180,E1 -26294.478,E2 -26294.478} C_VEL
LIN {X 0,Y 118.7,Z 228.372,A -85,B 0,C 180,E1 -26297.219,E2 -26297.219} C_VEL
LIN {X 0,Y 120.492,Z 230.518,A -85,B 0,C 180,E1 -26300.485,E2 -26300.485} C_VEL
LIN {X 0,Y 123.169,Z 235.8,A -85,B 0,C 180,E1 -26305.337,E2 -26305.337} C_VEL
LIN {X 0,Y 125.389,Z 241.171,A -85,B 0,C 180,E1 -26309.226,E2 -26309.226} C_VEL
LIN {X 0,Y 128.152,Z 249.485,A -85,B 0,C 180,E1 -26314.296,E2 -26314.296} C_VEL
LIN {X 0,Y 130.035,Z 256.968,A -85,B 0,C 180,E1 -26318.315,E2 -26318.315} C_VEL
LIN {X 0,Y 130.54,Z 261.036,A -85,B 0,C 180,E1 -26320.244,E2 -26320.244} C_VEL
LIN {X 0,Y 129.692,Z 269.311,A -85,B 0,C 180,E1 -26323.564,E2 -26323.564} C_VEL
LIN {X 0,Y 127.565,Z 279.111,A -85,B 0,C 180,E1 -26327.682,E2 -26327.682} C_VEL
LIN {X 0,Y 125.759,Z 284.275,A -85,B 0,C 180,E1 -26330.015,E2 -26330.015} C_VEL
LIN {X 0,Y 120.418,Z 293.275,A -85,B 0,C 180,E1 -26334.299,E2 -26334.299} C_VEL
LIN {X 0,Y 115.862,Z 300.527,A -85,B 0,C 180,E1 -26338.968,E2 -26338.968} C_VEL
LIN {X 0,Y 111.881,Z 306.314,A -85,B 0,C 180,E1 -26343.919,E2 -26343.919} C_VEL
LIN {X 0,Y 108.743,Z 310.87,A -85,B 0,C 180,E1 -26349.182,E2 -26349.182} C_VEL
LIN {X 0,Y 106.68,Z 314.342,A -85,B 0,C 180,E1 -26354.725,E2 -26354.725} C_VEL
LIN {X 0,Y 105.791,Z 316.075,A -85,B 0,C 180,E1 -26358.508,E2 -26358.508} C_VEL
LIN {X 0,Y 105.227,Z 317.397,A -85,B 0,C 180,E1 -26362.327,E2 -26362.327} C_VEL
LIN {X 0,Y 105.034,Z 318.326,A -85,B 0,C 180,E1 -26366.166,E2 -26366.166} C_VEL
LIN {X 0,Y 105.167,Z 318.85,A -85,B 0,C 180,E1 -26370.003,E2 -26370.003} C_VEL
LIN {X 0,Y 105.036,Z 318.926,A -85,B 0,C 180,E1 -26373.839,E2 -26373.839} C_VEL
LIN {X 0,Y 105.802,Z 317.922,A -85,B 0,C 180,E1 -26381.496,E2 -26381.496} C_VEL
LIN {X 0,Y 106.737,Z 316.833,A -85,B 0,C 180,E1 -26385.272,E2 -26385.272} C_VEL
LIN {X 0,Y 108.024,Z 315.294,A -85,B 0,C 180,E1 -26388.985,E2 -26388.985} C_VEL
LIN {X 0,Y 110.879,Z 312.211,A -85,B 0,C 180,E1 -26394.331,E2 -26394.331} C_VEL
LIN {X 0,Y 114.581,Z 308.08,A -85,B 0,C 180,E1 -26399.386,E2 -26399.386} C_VEL
LIN {X 0,Y 119.273,Z 302.633,A -85,B 0,C 180,E1 -26404.196,E2 -26404.196} C_VEL
LIN {X 0,Y 124.286,Z 296.155,A -85,B 0,C 180,E1 -26408.463,E2 -26408.463} C_VEL
LIN {X 0,Y 130.138,Z 287.933,A -85,B 0,C 180,E1 -26412.457,E2 -26412.457} C_VEL
LIN {X 0,Y 132.611,Z 280.921,A -85,B 0,C 180,E1 -26415.901,E2 -26415.901} C_VEL
LIN {X 0,Y 134.384,Z 274.102,A -85,B 0,C 180,E1 -26419.006,E2 -26419.006} C_VEL
LIN {X 0,Y 134.936,Z 271.073,A -85,B 0,C 180,E1 -26420.357,E2 -26420.357} C_VEL
LIN {X 0,Y 134.917,Z 267.41,A -85,B 0,C 180,E1 -26422.254,E2 -26422.254} C_VEL
LIN {X 0,Y 133.862,Z 260.133,A -85,B 0,C 180,E1 -26426.548,E2 -26426.548} C_VEL
LIN {X 0,Y 132.11,Z 252.879,A -85,B 0,C 180,E1 -26431.395,E2 -26431.395} C_VEL
LIN {X 0,Y 130.136,Z 246.854,A -85,B 0,C 180,E1 -26436.276,E2 -26436.276} C_VEL
LIN {X 0,Y 128.442,Z 242.214,A -85,B 0,C 180,E1 -26440.835,E2 -26440.835} C_VEL
LIN {X 0,Y 126.971,Z 238.472,A -85,B 0,C 180,E1 -26445.578,E2 -26445.578} C_VEL
LIN {X 0,Y 126.526,Z 237.515,A -85,B 0,C 180,E1 -26447.163,E2 -26447.163} C_VEL
LIN {X 0,Y 125.688,Z 236.227,A -85,B 0,C 180,E1 -26450.344,E2 -26450.344} C_VEL
LIN {X 0,Y 124.928,Z 233.932,A -85,B 0,C 180,E1 -26460.001,E2 -26460.001} C_VEL
LIN {X 0,Y 125.858,Z 236.463,A -85,B 0,C 180,E1 -26469.645,E2 -26469.645} C_VEL
LIN {X 0,Y 126.789,Z 237.714,A -85,B 0,C 180,E1 -26472.811,E2 -26472.811} C_VEL
LIN {X 0,Y 128.873,Z 242.092,A -85,B 0,C 180,E1 -26479.1,E2 -26479.1} C_VEL
LIN {X 0,Y 131.096,Z 246.873,A -85,B 0,C 180,E1 -26484.31,E2 -26484.31} C_VEL
LIN {X 0,Y 132.5,Z 250.208,A -85,B 0,C 180,E1 -26487.373,E2 -26487.373} C_VEL
LIN {X 0,Y 132.985,Z 253.5,A -85,B 0,C 180,E1 -26489.481,E2 -26489.481} C_VEL
LIN {X 0,Y 132.523,Z 258.814,A -85,B 0,C 180,E1 -26492.016,E2 -26492.016} C_VEL
LIN {X 0,Y 130.976,Z 265.925,A -85,B 0,C 180,E1 -26495.082,E2 -26495.082} C_VEL
LIN {X 0,Y 129.979,Z 271.185,A -85,B 0,C 180,E1 -26497.758,E2 -26497.758} C_VEL
LIN {X 0,Y 128.672,Z 278.266,A -85,B 0,C 180,E1 -26501.761,E2 -26501.761} C_VEL
LIN {X 0,Y 127.626,Z 281.149,A -85,B 0,C 180,E1 -26503.32,E2 -26503.32} C_VEL
LIN {X 0,Y 121.481,Z 289.49,A -85,B 0,C 180,E1 -26507.175,E2 -26507.175} C_VEL
LIN {X 0,Y 115.643,Z 296.34,A -85,B 0,C 180,E1 -26511.47,E2 -26511.47} C_VEL
LIN {X 0,Y 109.891,Z 302.615,A -85,B 0,C 180,E1 -26517.07,E2 -26517.07} C_VEL
LIN {X 0,Y 105.795,Z 306.715,A -85,B 0,C 180,E1 -26522.288,E2 -26522.288} C_VEL
LIN {X 0,Y 103.414,Z 308.877,A -85,B 0,C 180,E1 -26525.935,E2 -26525.935} C_VEL
LIN {X 0,Y 101.589,Z 310.558,A -85,B 0,C 180,E1 -26529.762,E2 -26529.762} C_VEL
LIN {X 0,Y 99.089,Z 312.725,A -85,B 0,C 180,E1 -26537.713,E2 -26537.713} C_VEL
LIN {X 0,Y 98.404,Z 313.209,A -85,B 0,C 180,E1 -26541.786,E2 -26541.786} C_VEL
LIN {X 0,Y 98.11,Z 313.275,A -85,B 0,C 180,E1 -26545.89,E2 -26545.89} C_VEL
LIN {X 0,Y 98.144,Z 312.964,A -85,B 0,C 180,E1 -26549.997,E2 -26549.997} C_VEL
LIN {X 0,Y 98.445,Z 312.277,A -85,B 0,C 180,E1 -26554.091,E2 -26554.091} C_VEL
LIN {X 0,Y 99.079,Z 311.193,A -85,B 0,C 180,E1 -26558.152,E2 -26558.152} C_VEL
LIN {X 0,Y 100.057,Z 309.669,A -85,B 0,C 180,E1 -26562.161,E2 -26562.161} C_VEL
LIN {X 0,Y 102.224,Z 306.614,A -85,B 0,C 180,E1 -26568.018,E2 -26568.018} C_VEL
LIN {X 0,Y 105.326,Z 302.511,A -85,B 0,C 180,E1 -26573.596,E2 -26573.596} C_VEL
LIN {X 0,Y 110.055,Z 296.239,A -85,B 0,C 180,E1 -26579.658,E2 -26579.658} C_VEL
LIN {X 0,Y 114.986,Z 289.406,A -85,B 0,C 180,E1 -26584.422,E2 -26584.422} C_VEL
LIN {X 0,Y 119.533,Z 282.428,A -85,B 0,C 180,E1 -26588.117,E2 -26588.117} C_VEL
LIN {X 0,Y 123.934,Z 274.828,A -85,B 0,C 180,E1 -26591.291,E2 -26591.291} C_VEL
LIN {X 0,Y 125.293,Z 267.18,A -85,B 0,C 180,E1 -26595.077,E2 -26595.077} C_VEL
LIN {X 0,Y 125.637,Z 261.661,A -85,B 0,C 180,E1 -26597.834,E2 -26597.834} C_VEL
LIN {X 0,Y 125.046,Z 256.456,A -85,B 0,C 180,E1 -26600.78,E2 -26600.78} C_VEL
LIN {X 0,Y 124.079,Z 252.096,A -85,B 0,C 180,E1 -26603.503,E2 -26603.503} C_VEL
LIN {X 0,Y 121.447,Z 245.491,A -85,B 0,C 180,E1 -26608.612,E2 -26608.612} C_VEL
LIN {X 0,Y 119.737,Z 241.765,A -85,B 0,C 180,E1 -26611.993,E2 -26611.993} C_VEL
LIN {X 0,Y 117.362,Z 237.009,A -85,B 0,C 180,E1 -26617.092,E2 -26617.092} C_VEL
LIN {X 0,Y 115.208,Z 233.625,A -85,B 0,C 180,E1 -26622.24,E2 -26622.24} C_VEL
LIN {X 0,Y 114.123,Z 231.727,A -85,B 0,C 180,E1 -26625.739,E2 -26625.739} C_VEL
LIN {X 0,Y 112.493,Z 228.24,A -85,B 0,C 180,E1 -26638.167,E2 -26638.167} C_VEL
LIN {X 0,Y 112.617,Z 227.959,A -85,B 0,C 180,E1 -26639.999,E2 -26639.999} C_VEL
LIN {X 0,Y 113.986,Z 231.401,A -85,B 0,C 180,E1 -26650.659,E2 -26650.659} C_VEL
LIN {X 0,Y 115.207,Z 232.821,A -85,B 0,C 180,E1 -26654.123,E2 -26654.123} C_VEL
LIN {X 0,Y 116.384,Z 235.492,A -85,B 0,C 180,E1 -26657.573,E2 -26657.573} C_VEL
LIN {X 0,Y 117.208,Z 236.517,A -85,B 0,C 180,E1 -26659.255,E2 -26659.255} C_VEL
LIN {X 0,Y 119.519,Z 241.513,A -85,B 0,C 180,E1 -26664.306,E2 -26664.306} C_VEL
LIN {X 0,Y 121.421,Z 247.183,A -85,B 0,C 180,E1 -26668.617,E2 -26668.617} C_VEL
LIN {X 0,Y 123.566,Z 254.91,A -85,B 0,C 180,E1 -26673.679,E2 -26673.679} C_VEL
LIN {X 0,Y 124.777,Z 261.368,A -85,B 0,C 180,E1 -26677.401,E2 -26677.401} C_VEL
LIN {X 0,Y 124.91,Z 265.097,A -85,B 0,C 180,E1 -26679.269,E2 -26679.269} C_VEL
LIN {X 0,Y 123.668,Z 272.323,A -85,B 0,C 180,E1 -26682.38,E2 -26682.38} C_VEL
LIN {X 0,Y 121.54,Z 280.404,A -85,B 0,C 180,E1 -26686.068,E2 -26686.068} C_VEL
LIN {X 0,Y 119.402,Z 285.604,A -85,B 0,C 180,E1 -26688.541,E2 -26688.541} C_VEL
LIN {X 0,Y 114.675,Z 292.984,A -85,B 0,C 180,E1 -26692.209,E2 -26692.209} C_VEL
LIN {X 0,Y 109.793,Z 300.253,A -85,B 0,C 180,E1 -26697.043,E2 -26697.043} C_VEL
LIN {X 0,Y 105.509,Z 306.058,A -85,B 0,C 180,E1 -26702.212,E2 -26702.212} C_VEL
LIN {X 0,Y 102.098,Z 310.628,A -85,B 0,C 180,E1 -26707.758,E2 -26707.758} C_VEL
LIN {X 0,Y 99.804,Z 314.11,A -85,B 0,C 180,E1 -26713.644,E2 -26713.644} C_VEL
LIN {X 0,Y 98.805,Z 315.852,A -85,B 0,C 180,E1 -26717.683,E2 -26717.683} C_VEL
LIN {X 0,Y 98.184,Z 317.181,A -85,B 0,C 180,E1 -26721.773,E2 -26721.773} C_VEL
LIN {X 0,Y 97.94,Z 318.114,A -85,B 0,C 180,E1 -26725.888,E2 -26725.888} C_VEL
LIN {X 0,Y 98.073,Z 318.648,A -85,B 0,C 180,E1 -26730.003,E2 -26730.003} C_VEL
LIN {X 0,Y 97.942,Z 318.731,A -85,B 0,C 180,E1 -26734.117,E2 -26734.117} C_VEL
LIN {X 0,Y 98.821,Z 317.737,A -85,B 0,C 180,E1 -26742.321,E2 -26742.321} C_VEL
LIN {X 0,Y 99.86,Z 316.656,A -85,B 0,C 180,E1 -26746.352,E2 -26746.352} C_VEL
LIN {X 0,Y 101.296,Z 315.125,A -85,B 0,C 180,E1 -26750.299,E2 -26750.299} C_VEL
LIN {X 0,Y 104.416,Z 312.054,A -85,B 0,C 180,E1 -26755.945,E2 -26755.945} C_VEL
LIN {X 0,Y 108.436,Z 307.936,A -85,B 0,C 180,E1 -26761.232,E2 -26761.232} C_VEL
LIN {X 0,Y 113.663,Z 302.165,A -85,B 0,C 180,E1 -26766.505,E2 -26766.505} C_VEL
LIN {X 0,Y 119.794,Z 294.805,A -85,B 0,C 180,E1 -26771.3,E2 -26771.3} C_VEL
LIN {X 0,Y 123.949,Z 289.323,A -85,B 0,C 180,E1 -26773.993,E2 -26773.993} C_VEL
LIN {X 0,Y 126.035,Z 284.635,A -85,B 0,C 180,E1 -26776.46,E2 -26776.46} C_VEL
LIN {X 0,Y 128.392,Z 277.489,A -85,B 0,C 180,E1 -26780.025,E2 -26780.025} C_VEL
LIN {X 0,Y 129.384,Z 272.832,A -85,B 0,C 180,E1 -26782.333,E2 -26782.333} C_VEL
LIN {X 0,Y 129.204,Z 268.201,A -85,B 0,C 180,E1 -26785.169,E2 -26785.169} C_VEL
LIN {X 0,Y 128.507,Z 262.944,A -85,B 0,C 180,E1 -26788.698,E2 -26788.698} C_VEL
LIN {X 0,Y 127.516,Z 257.473,A -85,B 0,C 180,E1 -26792.707,E2 -26792.707} C_VEL
LIN {X 0,Y 126.192,Z 252.509,A -85,B 0,C 180,E1 -26797.056,E2 -26797.056} C_VEL
LIN {X 0,Y 125.295,Z 249.235,A -85,B 0,C 180,E1 -26800.334,E2 -26800.334} C_VEL
LIN {X 0,Y 123.695,Z 244.314,A -85,B 0,C 180,E1 -26806.864,E2 -26806.864} C_VEL
LIN {X 0,Y 122.94,Z 242.898,A -85,B 0,C 180,E1 -26810.126,E2 -26810.126} C_VEL
LIN {X 0,Y 122.25,Z 240.557,A -85,B 0,C 180,E1 -26820.001,E2 -26820.001} C_VEL
LIN {X 0,Y 123.054,Z 243.084,A -85,B 0,C 180,E1 -26829.867,E2 -26829.867} C_VEL
LIN {X 0,Y 123.736,Z 244.631,A -85,B 0,C 180,E1 -26833.133,E2 -26833.133} C_VEL
LIN {X 0,Y 125.12,Z 247.71,A -85,B 0,C 180,E1 -26837.994,E2 -26837.994} C_VEL
LIN {X 0,Y 126.744,Z 251.716,A -85,B 0,C 180,E1 -26842.841,E2 -26842.841} C_VEL
LIN {X 0,Y 128.045,Z 255.297,A -85,B 0,C 180,E1 -26846.444,E2 -26846.444} C_VEL
LIN {X 0,Y 129.292,Z 261.224,A -85,B 0,C 180,E1 -26851.092,E2 -26851.092} C_VEL
LIN {X 0,Y 130.078,Z 268.075,A -85,B 0,C 180,E1 -26855.863,E2 -26855.863} C_VEL
LIN {X 0,Y 129.979,Z 271.185,A -85,B 0,C 180,E1 -26857.758,E2 -26857.758} C_VEL
LIN {X 0,Y 129.1,Z 273.844,A -85,B 0,C 180,E1 -26858.982,E2 -26858.982} C_VEL
LIN {X 0,Y 127.325,Z 276.676,A -85,B 0,C 180,E1 -26859.938,E2 -26859.938} C_VEL
LIN {X 0,Y 120.068,Z 285.013,A -85,B 0,C 180,E1 -26862.514,E2 -26862.514} C_VEL
LIN {X 0,Y 119.351,Z 285.874,A -85,B 0,C 180,E1 -26862.902,E2 -26862.902} C_VEL
LIN {X 0,Y 113.167,Z 293.22,A -85,B 0,C 180,E1 -26866.912,E2 -26866.912} C_VEL
LIN {X 0,Y 107.358,Z 299.371,A -85,B 0,C 180,E1 -26871.547,E2 -26871.547} C_VEL
LIN {X 0,Y 102.392,Z 304.244,A -85,B 0,C 180,E1 -26876.694,E2 -26876.694} C_VEL
LIN {X 0,Y 98.212,Z 307.997,A -85,B 0,C 180,E1 -26882.28,E2 -26882.28} C_VEL
LIN {X 0,Y 94.934,Z 310.73,A -85,B 0,C 180,E1 -26888.274,E2 -26888.274} C_VEL
LIN {X 0,Y 92.14,Z 312.909,A -85,B 0,C 180,E1 -26896.77,E2 -26896.77} C_VEL
LIN {X 0,Y 91.372,Z 313.403,A -85,B 0,C 180,E1 -26901.149,E2 -26901.149} C_VEL
LIN {X 0,Y 91.025,Z 313.475,A -85,B 0,C 180,E1 -26905.569,E2 -26905.569} C_VEL
LIN {X 0,Y 91.051,Z 313.17,A -85,B 0,C 180,E1 -26909.997,E2 -26909.997} C_VEL
LIN {X 0,Y 91.387,Z 312.488,A -85,B 0,C 180,E1 -26914.407,E2 -26914.407} C_VEL
LIN {X 0,Y 92.058,Z 311.415,A -85,B 0,C 180,E1 -26918.779,E2 -26918.779} C_VEL
LIN {X 0,Y 93.14,Z 309.898,A -85,B 0,C 180,E1 -26923.079,E2 -26923.079} C_VEL
LIN {X 0,Y 95.494,Z 306.856,A -85,B 0,C 180,E1 -26929.336,E2 -26929.336} C_VEL
LIN {X 0,Y 98.858,Z 302.766,A -85,B 0,C 180,E1 -26935.244,E2 -26935.244} C_VEL
LIN {X 0,Y 103.946,Z 296.508,A -85,B 0,C 180,E1 -26941.595,E2 -26941.595} C_VEL
LIN {X 0,Y 109.216,Z 289.69,A -85,B 0,C 180,E1 -26946.523,E2 -26946.523} C_VEL
LIN {X 0,Y 114.049,Z 282.73,A -85,B 0,C 180,E1 -26950.312,E2 -26950.312} C_VEL
LIN {X 0,Y 117.812,Z 276.808,A -85,B 0,C 180,E1 -26952.856,E2 -26952.856} C_VEL
LIN {X 0,Y 118.989,Z 272.51,A -85,B 0,C 180,E1 -26955.127,E2 -26955.127} C_VEL
LIN {X 0,Y 119.946,Z 266.953,A -85,B 0,C 180,E1 -26958.071,E2 -26958.071} C_VEL
LIN {X 0,Y 119.901,Z 261.763,A -85,B 0,C 180,E1 -26961.163,E2 -26961.163} C_VEL
LIN {X 0,Y 119.341,Z 257.571,A -85,B 0,C 180,E1 -26963.92,E2 -26963.92} C_VEL
LIN {X 0,Y 117.556,Z 252.048,A -85,B 0,C 180,E1 -26968.458,E2 -26968.458} C_VEL
LIN {X 0,Y 115.769,Z 247.354,A -85,B 0,C 180,E1 -26972.914,E2 -26972.914} C_VEL
LIN {X 0,Y 113.755,Z 242.831,A -85,B 0,C 180,E1 -26978.241,E2 -26978.241} C_VEL
LIN {X 0,Y 111.539,Z 238.618,A -85,B 0,C 180,E1 -26985.401,E2 -26985.401} C_VEL
LIN {X 0,Y 110.136,Z 236.385,A -85,B 0,C 180,E1 -26992.667,E2 -26992.667} C_VEL
LIN {X 0,Y 110.256,Z 234.775,A -85,B 0,C 180,E1 -26999.999,E2 -26999.999} C_VEL
LIN {X 0,Y 111.521,Z 238.197,A -85,B 0,C 180,E1 -27010.897,E2 -27010.897} C_VEL
LIN {X 0,Y 112.532,Z 240.031,A -85,B 0,C 180,E1 -27014.466,E2 -27014.466} C_VEL
LIN {X 0,Y 114.361,Z 243.741,A -85,B 0,C 180,E1 -27019.754,E2 -27019.754} C_VEL
LIN {X 0,Y 115.651,Z 247.102,A -85,B 0,C 180,E1 -27023.267,E2 -27023.267} C_VEL
LIN {X 0,Y 117.119,Z 252.554,A -85,B 0,C 180,E1 -27027.713,E2 -27027.713} C_VEL
LIN {X 0,Y 118.518,Z 258.932,A -85,B 0,C 180,E1 -27032.255,E2 -27032.255} C_VEL
LIN {X 0,Y 119.353,Z 264.981,A -85,B 0,C 180,E1 -27036.074,E2 -27036.074} C_VEL
LIN {X 0,Y 119.27,Z 268.263,A -85,B 0,C 180,E1 -27037.868,E2 -27037.868} C_VEL
LIN {X 0,Y 117.673,Z 275.183,A -85,B 0,C 180,E1 -27041.069,E2 -27041.069} C_VEL
LIN {X 0,Y 114.881,Z 283.64,A -85,B 0,C 180,E1 -27045.297,E2 -27045.297} C_VEL
LIN {X 0,Y 113.105,Z 286.92,A -85,B 0,C 180,E1 -27046.889,E2 -27046.889} C_VEL
LIN {X 0,Y 107.096,Z 295.542,A -85,B 0,C 180,E1 -27051.68,E2 -27051.68} C_VEL
LIN {X 0,Y 102.253,Z 302.046,A -85,B 0,C 180,E1 -27056.649,E2 -27056.649} C_VEL
LIN {X 0,Y 97.915,Z 307.435,A -85,B 0,C 180,E1 -27062.195,E2 -27062.195} C_VEL
LIN {X 0,Y 94.523,Z 311.641,A -85,B 0,C 180,E1 -27068.18,E2 -27068.18} C_VEL
LIN {X 0,Y 92.981,Z 313.878,A -85,B 0,C 180,E1 -27072.406,E2 -27072.406} C_VEL
LIN {X 0,Y 91.854,Z 315.629,A -85,B 0,C 180,E1 -27076.734,E2 -27076.734} C_VEL
LIN {X 0,Y 91.143,Z 316.963,A -85,B 0,C 180,E1 -27081.132,E2 -27081.132} C_VEL
LIN {X 0,Y 90.87,Z 317.903,A -85,B 0,C 180,E1 -27085.568,E2 -27085.568} C_VEL
LIN {X 0,Y 90.971,Z 318.445,A -85,B 0,C 180,E1 -27090.003,E2 -27090.003} C_VEL
LIN {X 0,Y 90.871,Z 318.536,A -85,B 0,C 180,E1 -27094.438,E2 -27094.438} C_VEL
LIN {X 0,Y 91.872,Z 317.552,A -85,B 0,C 180,E1 -27103.269,E2 -27103.269} C_VEL
LIN {X 0,Y 93.033,Z 316.478,A -85,B 0,C 180,E1 -27107.59,E2 -27107.59} C_VEL
LIN {X 0,Y 94.632,Z 314.956,A -85,B 0,C 180,E1 -27111.799,E2 -27111.799} C_VEL
LIN {X 0,Y 98.055,Z 311.897,A -85,B 0,C 180,E1 -27117.768,E2 -27117.768} C_VEL
LIN {X 0,Y 102.421,Z 307.791,A -85,B 0,C 180,E1 -27123.295,E2 -27123.295} C_VEL
LIN {X 0,Y 107.526,Z 302.559,A -85,B 0,C 180,E1 -27128.342,E2 -27128.342} C_VEL
LIN {X 0,Y 113.481,Z 295.923,A -85,B 0,C 180,E1 -27132.94,E2 -27132.94} C_VEL
LIN {X 0,Y 117.818,Z 290.69,A -85,B 0,C 180,E1 -27135.709,E2 -27135.709} C_VEL
LIN {X 0,Y 119.497,Z 287.724,A -85,B 0,C 180,E1 -27137.32,E2 -27137.32} C_VEL
LIN {X 0,Y 122.49,Z 280.285,A -85,B 0,C 180,E1 -27141.369,E2 -27141.369} C_VEL
LIN {X 0,Y 123.691,Z 276.194,A -85,B 0,C 180,E1 -27143.539,E2 -27143.539} C_VEL
LIN {X 0,Y 123.748,Z 270.575,A -85,B 0,C 180,E1 -27147.351,E2 -27147.351} C_VEL
LIN {X 0,Y 123.014,Z 263.479,A -85,B 0,C 180,E1 -27152.803,E2 -27152.803} C_VEL
LIN {X 0,Y 122.019,Z 257.981,A -85,B 0,C 180,E1 -27157.836,E2 -27157.836} C_VEL
LIN {X 0,Y 121.344,Z 254.669,A -85,B 0,C 180,E1 -27161.425,E2 -27161.425} C_VEL
LIN {X 0,Y 120.367,Z 251.069,A -85,B 0,C 180,E1 -27166.494,E2 -27166.494} C_VEL
LIN {X 0,Y 119.821,Z 249.426,A -85,B 0,C 180,E1 -27169.866,E2 -27169.866} C_VEL
LIN {X 0,Y 119.085,Z 247.66,A -85,B 0,C 180,E1 -27176.617,E2 -27176.617} C_VEL
LIN {X 0,Y 119.214,Z 247.029,A -85,B 0,C 180,E1 -27180.001,E2 -27180.001} C_VEL
LIN {X 0,Y 119.809,Z 249.588,A -85,B 0,C 180,E1 -27190.137,E2 -27190.137} C_VEL
LIN {X 0,Y 121.14,Z 253.211,A -85,B 0,C 180,E1 -27196.863,E2 -27196.863} C_VEL
LIN {X 0,Y 122.437,Z 257.005,A -85,B 0,C 180,E1 -27201.908,E2 -27201.908} C_VEL
LIN {X 0,Y 123.541,Z 260.881,A -85,B 0,C 180,E1 -27206.071,E2 -27206.071} C_VEL
LIN {X 0,Y 124.257,Z 266.287,A -85,B 0,C 180,E1 -27210.601,E2 -27210.601} C_VEL
LIN {X 0,Y 124.5,Z 272.454,A -85,B 0,C 180,E1 -27215.245,E2 -27215.245} C_VEL
LIN {X 0,Y 123.971,Z 275.938,A -85,B 0,C 180,E1 -27217.472,E2 -27217.472} C_VEL
LIN {X 0,Y 122.573,Z 281.12,A -85,B 0,C 180,E1 -27220.661,E2 -27220.661} C_VEL
LIN {X 0,Y 121.889,Z 282.578,A -85,B 0,C 180,E1 -27221.448,E2 -27221.448} C_VEL
LIN {X 0,Y 119.351,Z 285.874,A -85,B 0,C 180,E1 -27222.902,E2 -27222.902} C_VEL
LIN {X 0,Y 116.893,Z 288.352,A -85,B 0,C 180,E1 -27223.872,E2 -27223.872} C_VEL
LIN {X 0,Y 111.644,Z 292.108,A -85,B 0,C 180,E1 -27224.907,E2 -27224.907} C_VEL
LIN {X 0,Y 106.349,Z 295.607,A -85,B 0,C 180,E1 -27226.125,E2 -27226.125} C_VEL
LIN {X 0,Y 103.872,Z 297.591,A -85,B 0,C 180,E1 -27227.413,E2 -27227.413} C_VEL
LIN {X 0,Y 98.226,Z 302.898,A -85,B 0,C 180,E1 -27232.542,E2 -27232.542} C_VEL
LIN {X 0,Y 93.414,Z 307.024,A -85,B 0,C 180,E1 -27238.22,E2 -27238.22} C_VEL
LIN {X 0,Y 90.597,Z 309.207,A -85,B 0,C 180,E1 -27242.26,E2 -27242.26} C_VEL
LIN {X 0,Y 86.572,Z 312.193,A -85,B 0,C 180,E1 -27251.049,E2 -27251.049} C_VEL
LIN {X 0,Y 85.232,Z 313.093,A -85,B 0,C 180,E1 -27255.676,E2 -27255.676} C_VEL
LIN {X 0,Y 84.367,Z 313.597,A -85,B 0,C 180,E1 -27260.407,E2 -27260.407} C_VEL
LIN {X 0,Y 83.938,Z 313.676,A -85,B 0,C 180,E1 -27265.194,E2 -27265.194} C_VEL
LIN {X 0,Y 83.951,Z 313.376,A -85,B 0,C 180,E1 -27269.997,E2 -27269.997} C_VEL
LIN {X 0,Y 84.319,Z 312.7,A -85,B 0,C 180,E1 -27274.778,E2 -27274.778} C_VEL
LIN {X 0,Y 85.076,Z 311.635,A -85,B 0,C 180,E1 -27279.506,E2 -27279.506} C_VEL
LIN {X 0,Y 86.24,Z 310.127,A -85,B 0,C 180,E1 -27284.147,E2 -27284.147} C_VEL
LIN {X 0,Y 88.828,Z 307.098,A -85,B 0,C 180,E1 -27290.852,E2 -27290.852} C_VEL
LIN {X 0,Y 92.491,Z 303.021,A -85,B 0,C 180,E1 -27297.118,E2 -27297.118} C_VEL
LIN {X 0,Y 97.979,Z 296.777,A -85,B 0,C 180,E1 -27303.767,E2 -27303.767} C_VEL
LIN {X 0,Y 103.611,Z 289.974,A -85,B 0,C 180,E1 -27308.854,E2 -27308.854} C_VEL
LIN {X 0,Y 108.74,Z 283.032,A -85,B 0,C 180,E1 -27312.729,E2 -27312.729} C_VEL
LIN {X 0,Y 112.327,Z 277.607,A -85,B 0,C 180,E1 -27315.171,E2 -27315.171} C_VEL
LIN {X 0,Y 113.982,Z 271.555,A -85,B 0,C 180,E1 -27318.641,E2 -27318.641} C_VEL
LIN {X 0,Y 114.514,Z 267.619,A -85,B 0,C 180,E1 -27321.017,E2 -27321.017} C_VEL
LIN {X 0,Y 114.285,Z 262.408,A -85,B 0,C 180,E1 -27324.691,E2 -27324.691} C_VEL
LIN {X 0,Y 113.34,Z 258.329,A -85,B 0,C 180,E1 -27328.191,E2 -27328.191} C_VEL
LIN {X 0,Y 111.589,Z 252.805,A -85,B 0,C 180,E1 -27333.84,E2 -27333.84} C_VEL
LIN {X 0,Y 109.93,Z 248.5,A -85,B 0,C 180,E1 -27339.412,E2 -27339.412} C_VEL
LIN {X 0,Y 108.537,Z 245.358,A -85,B 0,C 180,E1 -27344.988,E2 -27344.988} C_VEL
LIN {X 0,Y 107.825,Z 243.97,A -85,B 0,C 180,E1 -27348.723,E2 -27348.723} C_VEL
LIN {X 0,Y 107.272,Z 242.051,A -85,B 0,C 180,E1 -27356.243,E2 -27356.243} C_VEL
LIN {X 0,Y 107.517,Z 241.443,A -85,B 0,C 180,E1 -27359.999,E2 -27359.999} C_VEL
LIN {X 0,Y 108.639,Z 244.919,A -85,B 0,C 180,E1 -27371.19,E2 -27371.19} C_VEL
LIN {X 0,Y 109.924,Z 247.887,A -85,B 0,C 180,E1 -27376.482,E2 -27376.482} C_VEL
LIN {X 0,Y 110.572,Z 249.27,A -85,B 0,C 180,E1 -27378.529,E2 -27378.529} C_VEL
LIN {X 0,Y 111.565,Z 252.546,A -85,B 0,C 180,E1 -27382.207,E2 -27382.207} C_VEL
LIN {X 0,Y 112.645,Z 257.876,A -85,B 0,C 180,E1 -27386.894,E2 -27386.894} C_VEL
LIN {X 0,Y 113.582,Z 264.229,A -85,B 0,C 180,E1 -27391.731,E2 -27391.731} C_VEL
LIN {X 0,Y 113.895,Z 269.653,A -85,B 0,C 180,E1 -27395.399,E2 -27395.399} C_VEL
LIN {X 0,Y 112.656,Z 274.842,A -85,B 0,C 180,E1 -27398.065,E2 -27398.065} C_VEL
LIN {X 0,Y 109.641,Z 283.313,A -85,B 0,C 180,E1 -27402.519,E2 -27402.519} C_VEL
LIN {X 0,Y 107.971,Z 286.614,A -85,B 0,C 180,E1 -27404.282,E2 -27404.282} C_VEL
LIN {X 0,Y 101.782,Z 295.012,A -85,B 0,C 180,E1 -27409.014,E2 -27409.014} C_VEL
LIN {X 0,Y 96.393,Z 301.781,A -85,B 0,C 180,E1 -27414.325,E2 -27414.325} C_VEL
LIN {X 0,Y 91.666,Z 307.182,A -85,B 0,C 180,E1 -27420.115,E2 -27420.115} C_VEL
LIN {X 0,Y 87.933,Z 311.401,A -85,B 0,C 180,E1 -27426.451,E2 -27426.451} C_VEL
LIN {X 0,Y 86.212,Z 313.646,A -85,B 0,C 180,E1 -27430.974,E2 -27430.974} C_VEL
LIN {X 0,Y 84.942,Z 315.406,A -85,B 0,C 180,E1 -27435.632,E2 -27435.632} C_VEL
LIN {X 0,Y 84.129,Z 316.747,A -85,B 0,C 180,E1 -27440.386,E2 -27440.386} C_VEL
LIN {X 0,Y 83.786,Z 317.692,A -85,B 0,C 180,E1 -27445.192,E2 -27445.192} C_VEL
LIN {X 0,Y 83.878,Z 318.242,A -85,B 0,C 180,E1 -27450.003,E2 -27450.003} C_VEL
LIN {X 0,Y 83.787,Z 318.341,A -85,B 0,C 180,E1 -27454.814,E2 -27454.814} C_VEL
LIN {X 0,Y 84.961,Z 317.367,A -85,B 0,C 180,E1 -27464.371,E2 -27464.371} C_VEL
LIN {X 0,Y 86.264,Z 316.3,A -85,B 0,C 180,E1 -27469.021,E2 -27469.021} C_VEL
LIN {X 0,Y 88.046,Z 314.787,A -85,B 0,C 180,E1 -27473.524,E2 -27473.524} C_VEL
LIN {X 0,Y 91.81,Z 311.74,A -85,B 0,C 180,E1 -27479.84,E2 -27479.84} C_VEL
LIN {X 0,Y 96.558,Z 307.648,A -85,B 0,C 180,E1 -27485.611,E2 -27485.611} C_VEL
LIN {X 0,Y 102.83,Z 301.63,A -85,B 0,C 180,E1 -27491.466,E2 -27491.466} C_VEL
LIN {X 0,Y 109.508,Z 294.574,A -85,B 0,C 180,E1 -27496.219,E2 -27496.219} C_VEL
LIN {X 0,Y 112.876,Z 290.582,A -85,B 0,C 180,E1 -27498.344,E2 -27498.344} C_VEL
LIN {X 0,Y 115.946,Z 284.443,A -85,B 0,C 180,E1 -27501.996,E2 -27501.996} C_VEL
LIN {X 0,Y 117.822,Z 279.824,A -85,B 0,C 180,E1 -27504.611,E2 -27504.611} C_VEL
LIN {X 0,Y 118.242,Z 277.331,A -85,B 0,C 180,E1 -27506.315,E2 -27506.315} C_VEL
LIN {X 0,Y 118.296,Z 271.826,A -85,B 0,C 180,E1 -27510.651,E2 -27510.651} C_VEL
LIN {X 0,Y 117.992,Z 266.473,A -85,B 0,C 180,E1 -27515.359,E2 -27515.359} C_VEL
LIN {X 0,Y 117.551,Z 262.974,A -85,B 0,C 180,E1 -27518.979,E2 -27518.979} C_VEL
LIN {X 0,Y 117.156,Z 259.961,A -85,B 0,C 180,E1 -27522.547,E2 -27522.547} C_VEL
LIN {X 0,Y 116.655,Z 257.626,A -85,B 0,C 180,E1 -27526.056,E2 -27526.056} C_VEL
LIN {X 0,Y 116.266,Z 255.804,A -85,B 0,C 180,E1 -27529.553,E2 -27529.553} C_VEL
LIN {X 0,Y 115.689,Z 253.933,A -85,B 0,C 180,E1 -27536.518,E2 -27536.518} C_VEL
LIN {X 0,Y 115.836,Z 253.309,A -85,B 0,C 180,E1 -27540.001,E2 -27540.001} C_VEL
LIN {X 0,Y 115.818,Z 255.104,A -85,B 0,C 180,E1 -27547.73,E2 -27547.73} C_VEL
LIN {X 0,Y 116.176,Z 255.947,A -85,B 0,C 180,E1 -27550.457,E2 -27550.457} C_VEL
LIN {X 0,Y 117.023,Z 258.772,A -85,B 0,C 180,E1 -27556.081,E2 -27556.081} C_VEL
LIN {X 0,Y 117.931,Z 262.136,A -85,B 0,C 180,E1 -27560.952,E2 -27560.952} C_VEL
LIN {X 0,Y 118.608,Z 265.07,A -85,B 0,C 180,E1 -27564.506,E2 -27564.506} C_VEL
LIN {X 0,Y 118.995,Z 270.029,A -85,B 0,C 180,E1 -27569.162,E2 -27569.162} C_VEL
LIN {X 0,Y 118.967,Z 274.913,A -85,B 0,C 180,E1 -27573.243,E2 -27573.243} C_VEL
LIN {X 0,Y 118.277,Z 278.653,A -85,B 0,C 180,E1 -27575.936,E2 -27575.936} C_VEL
LIN {X 0,Y 116.949,Z 282.677,A -85,B 0,C 180,E1 -27578.628,E2 -27578.628} C_VEL
LIN {X 0,Y 116.096,Z 284.154,A -85,B 0,C 180,E1 -27579.482,E2 -27579.482} C_VEL
LIN {X 0,Y 109.186,Z 292.169,A -85,B 0,C 180,E1 -27583.604,E2 -27583.604} C_VEL
LIN {X 0,Y 103.872,Z 297.591,A -85,B 0,C 180,E1 -27587.413,E2 -27587.413} C_VEL
LIN {X 0,Y 100.5,Z 300.42,A -85,B 0,C 180,E1 -27589.634,E2 -27589.634} C_VEL
LIN {X 0,Y 93.65,Z 304.594,A -85,B 0,C 180,E1 -27593.102,E2 -27593.102} C_VEL
LIN {X 0,Y 86.978,Z 307.979,A -85,B 0,C 180,E1 -27597.257,E2 -27597.257} C_VEL
LIN {X 0,Y 84.042,Z 309.572,A -85,B 0,C 180,E1 -27600.534,E2 -27600.534} C_VEL
LIN {X 0,Y 79.851,Z 312.372,A -85,B 0,C 180,E1 -27609.385,E2 -27609.385} C_VEL
LIN {X 0,Y 78.371,Z 313.277,A -85,B 0,C 180,E1 -27614.391,E2 -27614.391} C_VEL
LIN {X 0,Y 77.368,Z 313.79,A -85,B 0,C 180,E1 -27619.53,E2 -27619.53} C_VEL
LIN {X 0,Y 76.876,Z 313.877,A -85,B 0,C 180,E1 -27624.752,E2 -27624.752} C_VEL
LIN {X 0,Y 76.859,Z 313.582,A -85,B 0,C 180,E1 -27629.996,E2 -27629.996} C_VEL
LIN {X 0,Y 77.266,Z 312.911,A -85,B 0,C 180,E1 -27635.215,E2 -27635.215} C_VEL
LIN {X 0,Y 78.082,Z 311.856,A -85,B 0,C 180,E1 -27640.366,E2 -27640.366} C_VEL
LIN {X 0,Y 79.392,Z 310.356,A -85,B 0,C 180,E1 -27645.396,E2 -27645.396} C_VEL
LIN {X 0,Y 82.244,Z 307.339,A -85,B 0,C 180,E1 -27652.61,E2 -27652.61} C_VEL
LIN {X 0,Y 86.245,Z 303.275,A -85,B 0,C 180,E1 -27659.264,E2 -27659.264} C_VEL
LIN {X 0,Y 92.161,Z 297.045,A -85,B 0,C 180,E1 -27666.221,E2 -27666.221} C_VEL
LIN {X 0,Y 98.2,Z 290.258,A -85,B 0,C 180,E1 -27671.446,E2 -27671.446} C_VEL
LIN {X 0,Y 103.636,Z 283.334,A -85,B 0,C 180,E1 -27675.394,E2 -27675.394} C_VEL
LIN {X 0,Y 106.779,Z 278.915,A -85,B 0,C 180,E1 -27677.453,E2 -27677.453} C_VEL
LIN {X 0,Y 108.578,Z 273.244,A -85,B 0,C 180,E1 -27680.953,E2 -27680.953} C_VEL
LIN {X 0,Y 109.057,Z 269.482,A -85,B 0,C 180,E1 -27683.6,E2 -27683.6} C_VEL
LIN {X 0,Y 109.072,Z 266.632,A -85,B 0,C 180,E1 -27685.848,E2 -27685.848} C_VEL
LIN {X 0,Y 108.313,Z 262.447,A -85,B 0,C 180,E1 -27689.871,E2 -27689.871} C_VEL
LIN {X 0,Y 107.203,Z 258.101,A -85,B 0,C 180,E1 -27694.777,E2 -27694.777} C_VEL
LIN {X 0,Y 105.9,Z 254.012,A -85,B 0,C 180,E1 -27700.62,E2 -27700.62} C_VEL
LIN {X 0,Y 105.153,Z 251.97,A -85,B 0,C 180,E1 -27704.493,E2 -27704.493} C_VEL
LIN {X 0,Y 104.576,Z 250.399,A -85,B 0,C 180,E1 -27708.368,E2 -27708.368} C_VEL
LIN {X 0,Y 104.151,Z 248.519,A -85,B 0,C 180,E1 -27716.13,E2 -27716.13} C_VEL
LIN {X 0,Y 104.419,Z 247.943,A -85,B 0,C 180,E1 -27719.999,E2 -27719.999} C_VEL
LIN {X 0,Y 105.345,Z 251.453,A -85,B 0,C 180,E1 -27731.544,E2 -27731.544} C_VEL
LIN {X 0,Y 106.491,Z 254.546,A -85,B 0,C 180,E1 -27737.029,E2 -27737.029} C_VEL
LIN {X 0,Y 107.274,Z 257.836,A -85,B 0,C 180,E1 -27741.12,E2 -27741.12} C_VEL
LIN {X 0,Y 107.945,Z 263.054,A -85,B 0,C 180,E1 -27746.068,E2 -27746.068} C_VEL
LIN {X 0,Y 108.407,Z 269.367,A -85,B 0,C 180,E1 -27751.24,E2 -27751.24} C_VEL
LIN {X 0,Y 108.249,Z 273.225,A -85,B 0,C 180,E1 -27754.031,E2 -27754.031} C_VEL
LIN {X 0,Y 106.148,Z 279.373,A -85,B 0,C 180,E1 -27757.401,E2 -27757.401} C_VEL
LIN {X 0,Y 103.034,Z 286.303,A -85,B 0,C 180,E1 -27761.391,E2 -27761.391} C_VEL
LIN {X 0,Y 96.508,Z 294.73,A -85,B 0,C 180,E1 -27766.233,E2 -27766.233} C_VEL
LIN {X 0,Y 90.695,Z 301.514,A -85,B 0,C 180,E1 -27771.696,E2 -27771.696} C_VEL
LIN {X 0,Y 85.556,Z 306.929,A -85,B 0,C 180,E1 -27777.734,E2 -27777.734} C_VEL
LIN {X 0,Y 81.439,Z 311.16,A -85,B 0,C 180,E1 -27784.444,E2 -27784.444} C_VEL
LIN {X 0,Y 79.491,Z 313.412,A -85,B 0,C 180,E1 -27789.295,E2 -27789.295} C_VEL
LIN {X 0,Y 78.046,Z 315.183,A -85,B 0,C 180,E1 -27794.332,E2 -27794.332} C_VEL
LIN {X 0,Y 77.117,Z 316.529,A -85,B 0,C 180,E1 -27799.502,E2 -27799.502} C_VEL
LIN {X 0,Y 76.706,Z 317.48,A -85,B 0,C 180,E1 -27804.747,E2 -27804.747} C_VEL
LIN {X 0,Y 76.776,Z 318.038,A -85,B 0,C 180,E1 -27810.004,E2 -27810.004} C_VEL
LIN {X 0,Y 76.707,Z 318.145,A -85,B 0,C 180,E1 -27815.26,E2 -27815.26} C_VEL
LIN {X 0,Y 78.067,Z 317.181,A -85,B 0,C 180,E1 -27825.671,E2 -27825.671} C_VEL
LIN {X 0,Y 79.565,Z 316.121,A -85,B 0,C 180,E1 -27830.693,E2 -27830.693} C_VEL
LIN {X 0,Y 81.554,Z 314.618,A -85,B 0,C 180,E1 -27835.525,E2 -27835.525} C_VEL
LIN {X 0,Y 85.702,Z 311.584,A -85,B 0,C 180,E1 -27842.212,E2 -27842.212} C_VEL
LIN {X 0,Y 90.872,Z 307.504,A -85,B 0,C 180,E1 -27848.223,E2 -27848.223} C_VEL
LIN {X 0,Y 97.774,Z 301.326,A -85,B 0,C 180,E1 -27854.387,E2 -27854.387} C_VEL
LIN {X 0,Y 104.715,Z 294.459,A -85,B 0,C 180,E1 -27859.029,E2 -27859.029} C_VEL
LIN {X 0,Y 107.093,Z 291.834,A -85,B 0,C 180,E1 -27860.451,E2 -27860.451} C_VEL
LIN {X 0,Y 109.694,Z 287.514,A -85,B 0,C 180,E1 -27863.211,E2 -27863.211} C_VEL
LIN {X 0,Y 112.27,Z 282.31,A -85,B 0,C 180,E1 -27866.416,E2 -27866.416} C_VEL
LIN {X 0,Y 112.893,Z 277.791,A -85,B 0,C 180,E1 -27870.131,E2 -27870.131} C_VEL
LIN {X 0,Y 113.092,Z 273.32,A -85,B 0,C 180,E1 -27874.215,E2 -27874.215} C_VEL
LIN {X 0,Y 112.96,Z 268.87,A -85,B 0,C 180,E1 -27878.943,E2 -27878.943} C_VEL
LIN {X 0,Y 112.77,Z 265.177,A -85,B 0,C 180,E1 -27883.543,E2 -27883.543} C_VEL
LIN {X 0,Y 112.331,Z 262.019,A -85,B 0,C 180,E1 -27889.182,E2 -27889.182} C_VEL
LIN {X 0,Y 112.039,Z 260.794,A -85,B 0,C 180,E1 -27892.794,E2 -27892.794} C_VEL
LIN {X 0,Y 112.083,Z 259.387,A -85,B 0,C 180,E1 -27900.001,E2 -27900.001} C_VEL
LIN {X 0,Y 111.91,Z 261.114,A -85,B 0,C 180,E1 -27907.773,E2 -27907.773} C_VEL
LIN {X 0,Y 112.203,Z 262.095,A -85,B 0,C 180,E1 -27910.832,E2 -27910.832} C_VEL
LIN {X 0,Y 112.807,Z 264.984,A -85,B 0,C 180,E1 -27916.699,E2 -27916.699} C_VEL
LIN {X 0,Y 113.42,Z 268.462,A -85,B 0,C 180,E1 -27921.827,E2 -27921.827} C_VEL
LIN {X 0,Y 113.675,Z 269.895,A -85,B 0,C 180,E1 -27923.696,E2 -27923.696} C_VEL
LIN {X 0,Y 113.682,Z 273.674,A -85,B 0,C 180,E1 -27927.619,E2 -27927.619} C_VEL
LIN {X 0,Y 113.341,Z 278.195,A -85,B 0,C 180,E1 -27931.806,E2 -27931.806} C_VEL
LIN {X 0,Y 112.618,Z 281.135,A -85,B 0,C 180,E1 -27934.171,E2 -27934.171} C_VEL
LIN {X 0,Y 111.385,Z 284.254,A -85,B 0,C 180,E1 -27936.441,E2 -27936.441} C_VEL
LIN {X 0,Y 110.452,Z 285.73,A -85,B 0,C 180,E1 -27937.312,E2 -27937.312} C_VEL
LIN {X 0,Y 103.226,Z 293.46,A -85,B 0,C 180,E1 -27941.504,E2 -27941.504} C_VEL
LIN {X 0,Y 96.615,Z 299.639,A -85,B 0,C 180,E1 -27946.286,E2 -27946.286} C_VEL
LIN {X 0,Y 90.802,Z 304.54,A -85,B 0,C 180,E1 -27951.742,E2 -27951.742} C_VEL
LIN {X 0,Y 85.875,Z 308.318,A -85,B 0,C 180,E1 -27957.861,E2 -27957.861} C_VEL
LIN {X 0,Y 84.042,Z 309.572,A -85,B 0,C 180,E1 -27960.534,E2 -27960.534} C_VEL
LIN {X 0,Y 81.371,Z 311.005,A -85,B 0,C 180,E1 -27964.075,E2 -27964.075} C_VEL
